LIN {X 0,Y 496.716,Z 59.924,A -85,B 0,C 180,E1 24096.26,E2 24096.26} C_VEL
LIN {X 0,Y 496.76,Z 59.921,A -85,B 0,C 180,E1 24092.813,E2 24092.813} C_VEL
LIN {X 0,Y 496.725,Z 59.923,A -85,B 0,C 180,E1 24089.385,E2 24089.385} C_VEL
LIN {X 0,Y 496.699,Z 59.924,A -85,B 0,C 180,E1 24085.971,E2 24085.971} C_VEL
LIN {X 0,Y 496.701,Z 59.924,A -85,B 0,C 180,E1 24082.415,E2 24082.415} C_VEL
LIN {X 0,Y 496.743,Z 59.924,A -85,B 0,C 180,E1 24079.009,E2 24079.009} C_VEL
LIN {X 0,Y 496.74,Z 59.919,A -85,B 0,C 180,E1 24075.443,E2 24075.443} C_VEL
LIN {X 0,Y 496.703,Z 59.927,A -85,B 0,C 180,E1 24072.03,E2 24072.03} C_VEL
LIN {X 0,Y 496.702,Z 59.928,A -85,B 0,C 180,E1 24068.611,E2 24068.611} C_VEL
LIN {X 0,Y 496.775,Z 60.152,A -85,B 0,C 180,E1 24065.671,E2 24065.671} C_VEL
LIN {X 0,Y 502.744,Z 77.218,A -85,B 0,C 180,E1 24063.56,E2 24063.56} C_VEL
LIN {X 0,Y 505.317,Z 85.52,A -85,B 0,C 180,E1 24062.629,E2 24062.629} C_VEL
LIN {X 0,Y 502.906,Z 130.198,A -85,B 0,C 180,E1 24058.89,E2 24058.89} C_VEL
LIN {X 0,Y 501.717,Z 159.661,A -85,B 0,C 180,E1 24056.536,E2 24056.536} C_VEL
LIN {X 0,Y 503.214,Z 173.732,A -85,B 0,C 180,E1 24056.253,E2 24056.253} C_VEL
LIN {X 0,Y 501.873,Z 362.743,A -85,B 0,C 180,E1 24053.517,E2 24053.517} C_VEL
LIN {X 0,Y 501.376,Z 381.426,A -85,B 0,C 180,E1 24053.042,E2 24053.042} C_VEL
LIN {X 0,Y 500.757,Z 399.797,A -85,B 0,C 180,E1 24052.357,E2 24052.357} C_VEL
LIN {X 0,Y 500.08,Z 416.685,A -85,B 0,C 180,E1 24051.524,E2 24051.524} C_VEL
LIN {X 0,Y 499.326,Z 433.862,A -85,B 0,C 180,E1 24050.452,E2 24050.452} C_VEL
LIN {X 0,Y 498.576,Z 450.092,A -85,B 0,C 180,E1 24049.202,E2 24049.202} C_VEL
LIN {X 0,Y 497.872,Z 465.754,A -85,B 0,C 180,E1 24047.733,E2 24047.733} C_VEL
LIN {X 0,Y 497.273,Z 480.092,A -85,B 0,C 180,E1 24046.11,E2 24046.11} C_VEL
LIN {X 0,Y 496.822,Z 492.31,A -85,B 0,C 180,E1 24044.452,E2 24044.452} C_VEL
LIN {X 0,Y 496.496,Z 503.201,A -85,B 0,C 180,E1 24042.681,E2 24042.681} C_VEL
LIN {X 0,Y 496.273,Z 512.736,A -85,B 0,C 180,E1 24040.8,E2 24040.8} C_VEL
LIN {X 0,Y 496.163,Z 520.846,A -85,B 0,C 180,E1 24038.81,E2 24038.81} C_VEL
LIN {X 0,Y 496.121,Z 527.106,A -85,B 0,C 180,E1 24036.83,E2 24036.83} C_VEL
LIN {X 0,Y 496.12,Z 531.896,A -85,B 0,C 180,E1 24034.741,E2 24034.741} C_VEL
LIN {X 0,Y 496.135,Z 534.912,A -85,B 0,C 180,E1 24032.658,E2 24032.658} C_VEL
LIN {X 0,Y 496.149,Z 536.233,A -85,B 0,C 180,E1 24030.578,E2 24030.578} C_VEL
LIN {X 0,Y 496.141,Z 535.884,A -85,B 0,C 180,E1 24028.5,E2 24028.5} C_VEL
LIN {X 0,Y 496.114,Z 533.857,A -85,B 0,C 180,E1 24026.419,E2 24026.419} C_VEL
LIN {X 0,Y 496.098,Z 530.107,A -85,B 0,C 180,E1 24024.333,E2 24024.333} C_VEL
LIN {X 0,Y 496.123,Z 524.542,A -85,B 0,C 180,E1 24022.241,E2 24022.241} C_VEL
LIN {X 0,Y 496.195,Z 517.201,A -85,B 0,C 180,E1 24020.184,E2 24020.184} C_VEL
LIN {X 0,Y 496.361,Z 508.369,A -85,B 0,C 180,E1 24018.233,E2 24018.233} C_VEL
LIN {X 0,Y 496.659,Z 498.035,A -85,B 0,C 180,E1 24016.378,E2 24016.378} C_VEL
LIN {X 0,Y 497.07,Z 486.087,A -85,B 0,C 180,E1 24014.603,E2 24014.603} C_VEL
LIN {X 0,Y 497.658,Z 472.121,A -85,B 0,C 180,E1 24012.883,E2 24012.883} C_VEL
LIN {X 0,Y 498.316,Z 457.588,A -85,B 0,C 180,E1 24011.397,E2 24011.397} C_VEL
LIN {X 0,Y 499.047,Z 442.169,A -85,B 0,C 180,E1 24010.088,E2 24010.088} C_VEL
LIN {X 0,Y 499.804,Z 425.94,A -85,B 0,C 180,E1 24008.957,E2 24008.957} C_VEL
LIN {X 0,Y 500.54,Z 408.959,A -85,B 0,C 180,E1 24008.005,E2 24008.005} C_VEL
LIN {X 0,Y 501.216,Z 391.162,A -85,B 0,C 180,E1 24007.233,E2 24007.233} C_VEL
LIN {X 0,Y 501.791,Z 372.509,A -85,B 0,C 180,E1 24006.648,E2 24006.648} C_VEL
LIN {X 0,Y 502.171,Z 353.099,A -85,B 0,C 180,E1 24006.264,E2 24006.264} C_VEL
LIN {X 0,Y 503.355,Z 163.342,A -85,B 0,C 180,E1 24003.523,E2 24003.523} C_VEL
LIN {X 0,Y 502.895,Z 155.431,A -85,B 0,C 180,E1 24003.364,E2 24003.364} C_VEL
LIN {X 0,Y 505.189,Z 81.94,A -85,B 0,C 180,E1 23999.846,E2 23999.846} C_VEL
LIN {X 0,Y 496.866,Z 60.542,A -85,B 0,C 180,E1 23998.232,E2 23998.232} C_VEL
LIN {X 0,Y 496.764,Z 59.943,A -85,B 0,C 180,E1 23998.04,E2 23998.04} C_VEL
LIN {X 0,Y 496.765,Z 59.917,A -85,B 0,C 180,E1 23994.404,E2 23994.404} C_VEL
LIN {X 0,Y 496.767,Z 59.917,A -85,B 0,C 180,E1 23990.796,E2 23990.796} C_VEL
LIN {X 0,Y 496.755,Z 59.92,A -85,B 0,C 180,E1 23987.279,E2 23987.279} C_VEL
LIN {X 0,Y 496.762,Z 59.919,A -85,B 0,C 180,E1 23983.735,E2 23983.735} C_VEL
LIN {X 0,Y 496.767,Z 59.918,A -85,B 0,C 180,E1 23980.247,E2 23980.247} C_VEL
LIN {X 0,Y 496.768,Z 59.916,A -85,B 0,C 180,E1 23976.711,E2 23976.711} C_VEL
LIN {X 0,Y 496.761,Z 59.915,A -85,B 0,C 180,E1 23973.146,E2 23973.146} C_VEL
LIN {X 0,Y 496.749,Z 59.917,A -85,B 0,C 180,E1 23969.599,E2 23969.599} C_VEL
LIN {X 0,Y 496.754,Z 59.92,A -85,B 0,C 180,E1 23966.026,E2 23966.026} C_VEL
LIN {X 0,Y 496.774,Z 59.916,A -85,B 0,C 180,E1 23962.483,E2 23962.483} C_VEL
LIN {X 0,Y 496.77,Z 59.913,A -85,B 0,C 180,E1 23958.908,E2 23958.908} C_VEL
LIN {X 0,Y 496.768,Z 59.913,A -85,B 0,C 180,E1 23955.288,E2 23955.288} C_VEL
LIN {X 0,Y 496.746,Z 59.917,A -85,B 0,C 180,E1 23951.729,E2 23951.729} C_VEL
LIN {X 0,Y 496.742,Z 59.918,A -85,B 0,C 180,E1 23948.216,E2 23948.216} C_VEL
LIN {X 0,Y 496.761,Z 59.915,A -85,B 0,C 180,E1 23944.733,E2 23944.733} C_VEL
LIN {X 0,Y 496.773,Z 59.918,A -85,B 0,C 180,E1 23941.153,E2 23941.153} C_VEL
LIN {X 0,Y 496.763,Z 59.916,A -85,B 0,C 180,E1 23937.577,E2 23937.577} C_VEL
LIN {X 0,Y 496.737,Z 59.916,A -85,B 0,C 180,E1 23934.108,E2 23934.108} C_VEL
LIN {X 0,Y 496.732,Z 59.915,A -85,B 0,C 180,E1 23930.499,E2 23930.499} C_VEL
LIN {X 0,Y 496.748,Z 59.917,A -85,B 0,C 180,E1 23926.971,E2 23926.971} C_VEL
LIN {X 0,Y 496.772,Z 59.919,A -85,B 0,C 180,E1 23923.513,E2 23923.513} C_VEL
LIN {X 0,Y 496.754,Z 59.917,A -85,B 0,C 180,E1 23919.99,E2 23919.99} C_VEL
LIN {X 0,Y 496.729,Z 59.902,A -85,B 0,C 180,E1 23916.512,E2 23916.512} C_VEL
LIN {X 0,Y 496.728,Z 59.921,A -85,B 0,C 180,E1 23912.94,E2 23912.94} C_VEL
LIN {X 0,Y 496.754,Z 59.91,A -85,B 0,C 180,E1 23909.479,E2 23909.479} C_VEL
LIN {X 0,Y 496.768,Z 59.92,A -85,B 0,C 180,E1 23905.976,E2 23905.976} C_VEL
LIN {X 0,Y 496.741,Z 59.92,A -85,B 0,C 180,E1 23902.418,E2 23902.418} C_VEL
LIN {X 0,Y 496.719,Z 59.919,A -85,B 0,C 180,E1 23898.988,E2 23898.988} C_VEL
LIN {X 0,Y 496.724,Z 59.923,A -85,B 0,C 180,E1 23895.442,E2 23895.442} C_VEL
LIN {X 0,Y 496.765,Z 59.919,A -85,B 0,C 180,E1 23892.037,E2 23892.037} C_VEL
LIN {X 0,Y 496.741,Z 59.922,A -85,B 0,C 180,E1 23888.605,E2 23888.605} C_VEL
LIN {X 0,Y 496.76,Z 59.922,A -85,B 0,C 180,E1 23886.138,E2 23886.138} C_VEL
LIN {X 0,Y 496.526,Z 60.974,A -85,B 0,C 180,E1 23885.641,E2 23885.641} C_VEL
LIN {X 0,Y 495.866,Z 64.234,A -85,B 0,C 180,E1 23885.105,E2 23885.105} C_VEL
LIN {X 0,Y 493.642,Z 74.787,A -85,B 0,C 180,E1 23884.064,E2 23884.064} C_VEL
LIN {X 0,Y 492.439,Z 83.383,A -85,B 0,C 180,E1 23883.217,E2 23883.217} C_VEL
LIN {X 0,Y 492.424,Z 84.219,A -85,B 0,C 180,E1 23883.128,E2 23883.128} C_VEL
LIN {X 0,Y 492.207,Z 114.606,A -85,B 0,C 180,E1 23879.841,E2 23879.841} C_VEL
LIN {X 0,Y 491.855,Z 147.091,A -85,B 0,C 180,E1 23876.3,E2 23876.3} C_VEL
LIN {X 0,Y 491.542,Z 180.424,A -85,B 0,C 180,E1 23872.735,E2 23872.735} C_VEL
LIN {X 0,Y 491.569,Z 185.791,A -85,B 0,C 180,E1 23872.215,E2 23872.215} C_VEL
LIN {X 0,Y 492.039,Z 191.108,A -85,B 0,C 180,E1 23872.114,E2 23872.114} C_VEL
LIN {X 0,Y 491.357,Z 297.481,A -85,B 0,C 180,E1 23870.513,E2 23870.513} C_VEL
LIN {X 0,Y 491.296,Z 311.859,A -85,B 0,C 180,E1 23870.086,E2 23870.086} C_VEL
LIN {X 0,Y 491.08,Z 325.962,A -85,B 0,C 180,E1 23869.449,E2 23869.449} C_VEL
LIN {X 0,Y 490.712,Z 339.55,A -85,B 0,C 180,E1 23868.594,E2 23868.594} C_VEL
LIN {X 0,Y 490.308,Z 351.863,A -85,B 0,C 180,E1 23867.565,E2 23867.565} C_VEL
LIN {X 0,Y 489.912,Z 362.623,A -85,B 0,C 180,E1 23866.417,E2 23866.417} C_VEL
LIN {X 0,Y 489.49,Z 372.793,A -85,B 0,C 180,E1 23865.034,E2 23865.034} C_VEL
LIN {X 0,Y 489.123,Z 381.598,A -85,B 0,C 180,E1 23863.475,E2 23863.475} C_VEL
LIN {X 0,Y 488.845,Z 388.636,A -85,B 0,C 180,E1 23861.801,E2 23861.801} C_VEL
LIN {X 0,Y 488.666,Z 393.601,A -85,B 0,C 180,E1 23860.134,E2 23860.134} C_VEL
LIN {X 0,Y 488.558,Z 396.808,A -85,B 0,C 180,E1 23858.472,E2 23858.472} C_VEL
LIN {X 0,Y 488.503,Z 398.475,A -85,B 0,C 180,E1 23856.581,E2 23856.581} C_VEL
LIN {X 0,Y 488.508,Z 398.105,A -85,B 0,C 180,E1 23854.695,E2 23854.695} C_VEL
LIN {X 0,Y 488.575,Z 395.704,A -85,B 0,C 180,E1 23852.814,E2 23852.814} C_VEL
LIN {X 0,Y 488.708,Z 391.51,A -85,B 0,C 180,E1 23851.054,E2 23851.054} C_VEL
LIN {X 0,Y 488.893,Z 386.21,A -85,B 0,C 180,E1 23849.53,E2 23849.53} C_VEL
LIN {X 0,Y 489.189,Z 378.47,A -85,B 0,C 180,E1 23847.891,E2 23847.891} C_VEL
LIN {X 0,Y 489.571,Z 368.931,A -85,B 0,C 180,E1 23846.369,E2 23846.369} C_VEL
LIN {X 0,Y 489.993,Z 357.955,A -85,B 0,C 180,E1 23845.024,E2 23845.024} C_VEL
LIN {X 0,Y 490.361,Z 346.306,A -85,B 0,C 180,E1 23843.913,E2 23843.913} C_VEL
LIN {X 0,Y 490.725,Z 334.558,A -85,B 0,C 180,E1 23843.036,E2 23843.036} C_VEL
LIN {X 0,Y 491.017,Z 321.028,A -85,B 0,C 180,E1 23842.276,E2 23842.276} C_VEL
LIN {X 0,Y 491.145,Z 306.68,A -85,B 0,C 180,E1 23841.707,E2 23841.707} C_VEL
LIN {X 0,Y 491.164,Z 291.861,A -85,B 0,C 180,E1 23841.346,E2 23841.346} C_VEL
LIN {X 0,Y 491.891,Z 181.867,A -85,B 0,C 180,E1 23839.725,E2 23839.725} C_VEL
LIN {X 0,Y 492.368,Z 131.209,A -85,B 0,C 180,E1 23836.494,E2 23836.494} C_VEL
LIN {X 0,Y 492.96,Z 86.133,A -85,B 0,C 180,E1 23833.533,E2 23833.533} C_VEL
LIN {X 0,Y 493.461,Z 85.428,A -85,B 0,C 180,E1 23833.338,E2 23833.338} C_VEL
LIN {X 0,Y 495.053,Z 86.354,A -85,B 0,C 180,E1 23833.122,E2 23833.122} C_VEL
LIN {X 0,Y 493.208,Z 136.927,A -85,B 0,C 180,E1 23829.406,E2 23829.406} C_VEL
LIN {X 0,Y 492.18,Z 171.769,A -85,B 0,C 180,E1 23826.9,E2 23826.9} C_VEL
LIN {X 0,Y 493.337,Z 184.723,A -85,B 0,C 180,E1 23826.64,E2 23826.64} C_VEL
LIN {X 0,Y 492.138,Z 292.661,A -85,B 0,C 180,E1 23824.909,E2 23824.909} C_VEL
LIN {X 0,Y 491.908,Z 307.221,A -85,B 0,C 180,E1 23824.474,E2 23824.474} C_VEL
LIN {X 0,Y 491.557,Z 320.784,A -85,B 0,C 180,E1 23823.872,E2 23823.872} C_VEL
LIN {X 0,Y 491.096,Z 334.583,A -85,B 0,C 180,E1 23823.043,E2 23823.043} C_VEL
LIN {X 0,Y 490.581,Z 347.204,A -85,B 0,C 180,E1 23822.045,E2 23822.045} C_VEL
LIN {X 0,Y 490.103,Z 358.821,A -85,B 0,C 180,E1 23820.879,E2 23820.879} C_VEL
LIN {X 0,Y 489.623,Z 369.502,A -85,B 0,C 180,E1 23819.516,E2 23819.516} C_VEL
LIN {X 0,Y 489.213,Z 378.649,A -85,B 0,C 180,E1 23818.015,E2 23818.015} C_VEL
LIN {X 0,Y 488.922,Z 385.866,A -85,B 0,C 180,E1 23816.484,E2 23816.484} C_VEL
LIN {X 0,Y 488.704,Z 391.966,A -85,B 0,C 180,E1 23814.72,E2 23814.72} C_VEL
LIN {X 0,Y 488.576,Z 396.002,A -85,B 0,C 180,E1 23812.952,E2 23812.952} C_VEL
LIN {X 0,Y 488.519,Z 398.188,A -85,B 0,C 180,E1 23811.222,E2 23811.222} C_VEL
LIN {X 0,Y 488.523,Z 398.654,A -85,B 0,C 180,E1 23809.394,E2 23809.394} C_VEL
LIN {X 0,Y 488.582,Z 397.307,A -85,B 0,C 180,E1 23807.627,E2 23807.627} C_VEL
LIN {X 0,Y 488.713,Z 394.286,A -85,B 0,C 180,E1 23805.899,E2 23805.899} C_VEL
LIN {X 0,Y 488.92,Z 389.202,A -85,B 0,C 180,E1 23804.126,E2 23804.126} C_VEL
LIN {X 0,Y 489.201,Z 382.95,A -85,B 0,C 180,E1 23802.573,E2 23802.573} C_VEL
LIN {X 0,Y 489.611,Z 374.598,A -85,B 0,C 180,E1 23801.001,E2 23801.001} C_VEL
LIN {X 0,Y 490.115,Z 364.396,A -85,B 0,C 180,E1 23799.531,E2 23799.531} C_VEL
LIN {X 0,Y 490.644,Z 353.329,A -85,B 0,C 180,E1 23798.281,E2 23798.281} C_VEL
LIN {X 0,Y 491.202,Z 341.189,A -85,B 0,C 180,E1 23797.197,E2 23797.197} C_VEL
LIN {X 0,Y 491.738,Z 327.186,A -85,B 0,C 180,E1 23796.241,E2 23796.241} C_VEL
LIN {X 0,Y 492.164,Z 313.062,A -85,B 0,C 180,E1 23795.523,E2 23795.523} C_VEL
LIN {X 0,Y 492.489,Z 297.592,A -85,B 0,C 180,E1 23794.979,E2 23794.979} C_VEL
LIN {X 0,Y 492.743,Z 277.093,A -85,B 0,C 180,E1 23794.576,E2 23794.576} C_VEL
LIN {X 0,Y 493.812,Z 188.367,A -85,B 0,C 180,E1 23793.093,E2 23793.093} C_VEL
LIN {X 0,Y 491.269,Z 174.322,A -85,B 0,C 180,E1 23792.689,E2 23792.689} C_VEL
LIN {X 0,Y 492.482,Z 144.862,A -85,B 0,C 180,E1 23789.028,E2 23789.028} C_VEL
LIN {X 0,Y 493.866,Z 117.28,A -85,B 0,C 180,E1 23785.546,E2 23785.546} C_VEL
LIN {X 0,Y 495.5,Z 87.632,A -85,B 0,C 180,E1 23781.733,E2 23781.733} C_VEL
LIN {X 0,Y 495.539,Z 84.368,A -85,B 0,C 180,E1 23781.297,E2 23781.297} C_VEL
LIN {X 0,Y 491.064,Z 68.425,A -85,B 0,C 180,E1 23778.766,E2 23778.766} C_VEL
LIN {X 0,Y 488.818,Z 61.026,A -85,B 0,C 180,E1 23777.483,E2 23777.483} C_VEL
LIN {X 0,Y 488.832,Z 60.909,A -85,B 0,C 180,E1 23773.967,E2 23773.967} C_VEL
LIN {X 0,Y 488.822,Z 60.908,A -85,B 0,C 180,E1 23770.37,E2 23770.37} C_VEL
LIN {X 0,Y 488.787,Z 60.91,A -85,B 0,C 180,E1 23766.932,E2 23766.932} C_VEL
LIN {X 0,Y 488.781,Z 60.912,A -85,B 0,C 180,E1 23763.381,E2 23763.381} C_VEL
LIN {X 0,Y 488.797,Z 60.911,A -85,B 0,C 180,E1 23759.883,E2 23759.883} C_VEL
LIN {X 0,Y 488.824,Z 60.91,A -85,B 0,C 180,E1 23756.365,E2 23756.365} C_VEL
LIN {X 0,Y 488.807,Z 60.91,A -85,B 0,C 180,E1 23752.832,E2 23752.832} C_VEL
LIN {X 0,Y 488.774,Z 60.911,A -85,B 0,C 180,E1 23749.391,E2 23749.391} C_VEL
LIN {X 0,Y 488.77,Z 60.91,A -85,B 0,C 180,E1 23745.79,E2 23745.79} C_VEL
LIN {X 0,Y 488.799,Z 60.91,A -85,B 0,C 180,E1 23742.378,E2 23742.378} C_VEL
LIN {X 0,Y 488.827,Z 60.908,A -85,B 0,C 180,E1 23738.775,E2 23738.775} C_VEL
LIN {X 0,Y 488.79,Z 60.911,A -85,B 0,C 180,E1 23735.263,E2 23735.263} C_VEL
LIN {X 0,Y 488.765,Z 60.912,A -85,B 0,C 180,E1 23731.8,E2 23731.8} C_VEL
LIN {X 0,Y 488.761,Z 60.913,A -85,B 0,C 180,E1 23728.144,E2 23728.144} C_VEL
LIN {X 0,Y 488.787,Z 60.913,A -85,B 0,C 180,E1 23724.705,E2 23724.705} C_VEL
LIN {X 0,Y 488.816,Z 60.912,A -85,B 0,C 180,E1 23721.199,E2 23721.199} C_VEL
LIN {X 0,Y 488.765,Z 60.915,A -85,B 0,C 180,E1 23717.777,E2 23717.777} C_VEL
LIN {X 0,Y 488.758,Z 60.915,A -85,B 0,C 180,E1 23714.275,E2 23714.275} C_VEL
LIN {X 0,Y 488.77,Z 60.915,A -85,B 0,C 180,E1 23710.736,E2 23710.736} C_VEL
LIN {X 0,Y 488.817,Z 60.908,A -85,B 0,C 180,E1 23707.41,E2 23707.41} C_VEL
LIN {X 0,Y 488.795,Z 61.141,A -85,B 0,C 180,E1 23706.24,E2 23706.24} C_VEL
LIN {X 0,Y 494.085,Z 75.723,A -85,B 0,C 180,E1 23704.345,E2 23704.345} C_VEL
LIN {X 0,Y 498.039,Z 88.036,A -85,B 0,C 180,E1 23702.899,E2 23702.899} C_VEL
LIN {X 0,Y 495.366,Z 133.317,A -85,B 0,C 180,E1 23699.041,E2 23699.041} C_VEL
LIN {X 0,Y 494.195,Z 159.804,A -85,B 0,C 180,E1 23696.886,E2 23696.886} C_VEL
LIN {X 0,Y 495.772,Z 174.654,A -85,B 0,C 180,E1 23696.58,E2 23696.58} C_VEL
LIN {X 0,Y 494.31,Z 362.064,A -85,B 0,C 180,E1 23693.828,E2 23693.828} C_VEL
LIN {X 0,Y 493.779,Z 380.78,A -85,B 0,C 180,E1 23693.345,E2 23693.345} C_VEL
LIN {X 0,Y 493.115,Z 398.948,A -85,B 0,C 180,E1 23692.66,E2 23692.66} C_VEL
LIN {X 0,Y 492.342,Z 416.524,A -85,B 0,C 180,E1 23691.776,E2 23691.776} C_VEL
LIN {X 0,Y 491.555,Z 433.003,A -85,B 0,C 180,E1 23690.728,E2 23690.728} C_VEL
LIN {X 0,Y 490.75,Z 449.218,A -85,B 0,C 180,E1 23689.459,E2 23689.459} C_VEL
LIN {X 0,Y 489.979,Z 465.054,A -85,B 0,C 180,E1 23687.947,E2 23687.947} C_VEL
LIN {X 0,Y 489.363,Z 478.705,A -85,B 0,C 180,E1 23686.378,E2 23686.378} C_VEL
LIN {X 0,Y 488.868,Z 491.134,A -85,B 0,C 180,E1 23684.669,E2 23684.669} C_VEL
LIN {X 0,Y 488.526,Z 501.928,A -85,B 0,C 180,E1 23682.891,E2 23682.891} C_VEL
LIN {X 0,Y 488.294,Z 511.506,A -85,B 0,C 180,E1 23680.979,E2 23680.979} C_VEL
LIN {X 0,Y 488.195,Z 519.655,A -85,B 0,C 180,E1 23678.955,E2 23678.955} C_VEL
LIN {X 0,Y 488.165,Z 525.946,A -85,B 0,C 180,E1 23676.942,E2 23676.942} C_VEL
LIN {X 0,Y 488.18,Z 530.761,A -85,B 0,C 180,E1 23674.818,E2 23674.818} C_VEL
LIN {X 0,Y 488.206,Z 533.796,A -85,B 0,C 180,E1 23672.701,E2 23672.701} C_VEL
LIN {X 0,Y 488.225,Z 535.128,A -85,B 0,C 180,E1 23670.588,E2 23670.588} C_VEL
LIN {X 0,Y 488.215,Z 534.781,A -85,B 0,C 180,E1 23668.475,E2 23668.475} C_VEL
LIN {X 0,Y 488.179,Z 532.751,A -85,B 0,C 180,E1 23666.361,E2 23666.361} C_VEL
LIN {X 0,Y 488.15,Z 528.992,A -85,B 0,C 180,E1 23664.241,E2 23664.241} C_VEL
LIN {X 0,Y 488.156,Z 523.411,A -85,B 0,C 180,E1 23662.113,E2 23662.113} C_VEL
LIN {X 0,Y 488.214,Z 516.331,A -85,B 0,C 180,E1 23660.091,E2 23660.091} C_VEL
LIN {X 0,Y 488.385,Z 507.338,A -85,B 0,C 180,E1 23658.068,E2 23658.068} C_VEL
LIN {X 0,Y 488.697,Z 496.822,A -85,B 0,C 180,E1 23656.151,E2 23656.151} C_VEL
LIN {X 0,Y 489.158,Z 484.562,A -85,B 0,C 180,E1 23654.311,E2 23654.311} C_VEL
LIN {X 0,Y 489.791,Z 470.803,A -85,B 0,C 180,E1 23652.6,E2 23652.6} C_VEL
LIN {X 0,Y 490.509,Z 456.185,A -85,B 0,C 180,E1 23651.09,E2 23651.09} C_VEL
LIN {X 0,Y 491.31,Z 440.484,A -85,B 0,C 180,E1 23649.747,E2 23649.747} C_VEL
LIN {X 0,Y 492.172,Z 423.339,A -85,B 0,C 180,E1 23648.552,E2 23648.552} C_VEL
LIN {X 0,Y 492.983,Z 405.873,A -85,B 0,C 180,E1 23647.587,E2 23647.587} C_VEL
LIN {X 0,Y 493.729,Z 387.328,A -85,B 0,C 180,E1 23646.811,E2 23646.811} C_VEL
LIN {X 0,Y 494.323,Z 368.66,A -85,B 0,C 180,E1 23646.26,E2 23646.26} C_VEL
LIN {X 0,Y 494.652,Z 348.014,A -85,B 0,C 180,E1 23645.887,E2 23645.887} C_VEL
LIN {X 0,Y 495.912,Z 163.899,A -85,B 0,C 180,E1 23643.19,E2 23643.19} C_VEL
LIN {X 0,Y 495.447,Z 155.03,A -85,B 0,C 180,E1 23642.996,E2 23642.996} C_VEL
LIN {X 0,Y 497.86,Z 84.428,A -85,B 0,C 180,E1 23639.555,E2 23639.555} C_VEL
LIN {X 0,Y 488.912,Z 61.44,A -85,B 0,C 180,E1 23637.776,E2 23637.776} C_VEL
LIN {X 0,Y 488.832,Z 60.926,A -85,B 0,C 180,E1 23637.597,E2 23637.597} C_VEL
LIN {X 0,Y 488.823,Z 60.909,A -85,B 0,C 180,E1 23634.054,E2 23634.054} C_VEL
LIN {X 0,Y 488.83,Z 60.907,A -85,B 0,C 180,E1 23630.454,E2 23630.454} C_VEL
LIN {X 0,Y 488.823,Z 60.906,A -85,B 0,C 180,E1 23626.905,E2 23626.905} C_VEL
LIN {X 0,Y 488.815,Z 60.907,A -85,B 0,C 180,E1 23623.268,E2 23623.268} C_VEL
LIN {X 0,Y 488.816,Z 60.909,A -85,B 0,C 180,E1 23619.657,E2 23619.657} C_VEL
LIN {X 0,Y 488.828,Z 60.908,A -85,B 0,C 180,E1 23616.092,E2 23616.092} C_VEL
LIN {X 0,Y 488.828,Z 60.907,A -85,B 0,C 180,E1 23612.544,E2 23612.544} C_VEL
LIN {X 0,Y 488.833,Z 60.903,A -85,B 0,C 180,E1 23608.908,E2 23608.908} C_VEL
LIN {X 0,Y 488.82,Z 60.904,A -85,B 0,C 180,E1 23605.303,E2 23605.303} C_VEL
LIN {X 0,Y 488.807,Z 60.907,A -85,B 0,C 180,E1 23601.73,E2 23601.73} C_VEL
LIN {X 0,Y 488.809,Z 60.908,A -85,B 0,C 180,E1 23598.114,E2 23598.114} C_VEL
LIN {X 0,Y 488.831,Z 60.903,A -85,B 0,C 180,E1 23594.571,E2 23594.571} C_VEL
LIN {X 0,Y 488.831,Z 60.907,A -85,B 0,C 180,E1 23590.959,E2 23590.959} C_VEL
LIN {X 0,Y 488.835,Z 60.903,A -85,B 0,C 180,E1 23587.285,E2 23587.285} C_VEL
LIN {X 0,Y 488.809,Z 60.902,A -85,B 0,C 180,E1 23583.753,E2 23583.753} C_VEL
LIN {X 0,Y 488.798,Z 60.901,A -85,B 0,C 180,E1 23580.234,E2 23580.234} C_VEL
LIN {X 0,Y 488.81,Z 60.908,A -85,B 0,C 180,E1 23576.716,E2 23576.716} C_VEL
LIN {X 0,Y 488.838,Z 60.907,A -85,B 0,C 180,E1 23573.187,E2 23573.187} C_VEL
LIN {X 0,Y 488.828,Z 60.9,A -85,B 0,C 180,E1 23569.63,E2 23569.63} C_VEL
LIN {X 0,Y 488.798,Z 60.902,A -85,B 0,C 180,E1 23566.153,E2 23566.153} C_VEL
LIN {X 0,Y 488.791,Z 60.905,A -85,B 0,C 180,E1 23562.623,E2 23562.623} C_VEL
LIN {X 0,Y 488.807,Z 60.907,A -85,B 0,C 180,E1 23559.15,E2 23559.15} C_VEL
LIN {X 0,Y 488.831,Z 60.889,A -85,B 0,C 180,E1 23555.724,E2 23555.724} C_VEL
LIN {X 0,Y 488.808,Z 60.907,A -85,B 0,C 180,E1 23552.2,E2 23552.2} C_VEL
LIN {X 0,Y 488.784,Z 60.904,A -85,B 0,C 180,E1 23548.763,E2 23548.763} C_VEL
LIN {X 0,Y 488.788,Z 60.903,A -85,B 0,C 180,E1 23545.199,E2 23545.199} C_VEL
LIN {X 0,Y 488.818,Z 60.912,A -85,B 0,C 180,E1 23541.7,E2 23541.7} C_VEL
LIN {X 0,Y 488.83,Z 60.907,A -85,B 0,C 180,E1 23538.116,E2 23538.116} C_VEL
LIN {X 0,Y 488.802,Z 60.91,A -85,B 0,C 180,E1 23534.555,E2 23534.555} C_VEL
LIN {X 0,Y 488.775,Z 60.913,A -85,B 0,C 180,E1 23531.043,E2 23531.043} C_VEL
LIN {X 0,Y 488.777,Z 60.916,A -85,B 0,C 180,E1 23527.411,E2 23527.411} C_VEL
LIN {X 0,Y 488.827,Z 61.168,A -85,B 0,C 180,E1 23525.781,E2 23525.781} C_VEL
LIN {X 0,Y 492.431,Z 75.428,A -85,B 0,C 180,E1 23524.062,E2 23524.062} C_VEL
LIN {X 0,Y 492.424,Z 84.219,A -85,B 0,C 180,E1 23523.128,E2 23523.128} C_VEL
LIN {X 0,Y 491.471,Z 90.111,A -85,B 0,C 180,E1 23522.55,E2 23522.55} C_VEL
LIN {X 0,Y 485.216,Z 107.25,A -85,B 0,C 180,E1 23521.027,E2 23521.027} C_VEL
LIN {X 0,Y 484.662,Z 111.429,A -85,B 0,C 180,E1 23520.597,E2 23520.597} C_VEL
LIN {X 0,Y 484.302,Z 143.545,A -85,B 0,C 180,E1 23517.078,E2 23517.078} C_VEL
LIN {X 0,Y 483.926,Z 176.363,A -85,B 0,C 180,E1 23513.548,E2 23513.548} C_VEL
LIN {X 0,Y 483.915,Z 186.439,A -85,B 0,C 180,E1 23512.511,E2 23512.511} C_VEL
LIN {X 0,Y 484.433,Z 191.716,A -85,B 0,C 180,E1 23512.399,E2 23512.399} C_VEL
LIN {X 0,Y 483.702,Z 298.42,A -85,B 0,C 180,E1 23510.77,E2 23510.77} C_VEL
LIN {X 0,Y 483.639,Z 312.821,A -85,B 0,C 180,E1 23510.338,E2 23510.338} C_VEL
LIN {X 0,Y 483.415,Z 326.772,A -85,B 0,C 180,E1 23509.701,E2 23509.701} C_VEL
LIN {X 0,Y 483.024,Z 340.331,A -85,B 0,C 180,E1 23508.838,E2 23508.838} C_VEL
LIN {X 0,Y 482.586,Z 352.724,A -85,B 0,C 180,E1 23507.793,E2 23507.793} C_VEL
LIN {X 0,Y 482.156,Z 363.533,A -85,B 0,C 180,E1 23506.628,E2 23506.628} C_VEL
LIN {X 0,Y 481.712,Z 373.35,A -85,B 0,C 180,E1 23505.283,E2 23505.283} C_VEL
LIN {X 0,Y 481.322,Z 381.658,A -85,B 0,C 180,E1 23503.82,E2 23503.82} C_VEL
LIN {X 0,Y 481.02,Z 388.542,A -85,B 0,C 180,E1 23502.24,E2 23502.24} C_VEL
LIN {X 0,Y 480.803,Z 393.911,A -85,B 0,C 180,E1 23500.544,E2 23500.544} C_VEL
LIN {X 0,Y 480.656,Z 397.602,A -85,B 0,C 180,E1 23498.733,E2 23498.733} C_VEL
LIN {X 0,Y 480.585,Z 399.41,A -85,B 0,C 180,E1 23496.93,E2 23496.93} C_VEL
LIN {X 0,Y 480.573,Z 399.446,A -85,B 0,C 180,E1 23495.132,E2 23495.132} C_VEL
LIN {X 0,Y 480.626,Z 397.72,A -85,B 0,C 180,E1 23493.338,E2 23493.338} C_VEL
LIN {X 0,Y 480.762,Z 393.835,A -85,B 0,C 180,E1 23491.429,E2 23491.429} C_VEL
LIN {X 0,Y 480.972,Z 388.092,A -85,B 0,C 180,E1 23489.642,E2 23489.642} C_VEL
LIN {X 0,Y 481.251,Z 381.205,A -85,B 0,C 180,E1 23488.094,E2 23488.094} C_VEL
LIN {X 0,Y 481.607,Z 372.979,A -85,B 0,C 180,E1 23486.667,E2 23486.667} C_VEL
LIN {X 0,Y 482.053,Z 362.367,A -85,B 0,C 180,E1 23485.24,E2 23485.24} C_VEL
LIN {X 0,Y 482.488,Z 350.344,A -85,B 0,C 180,E1 23483.992,E2 23483.992} C_VEL
LIN {X 0,Y 482.896,Z 337.65,A -85,B 0,C 180,E1 23482.982,E2 23482.982} C_VEL
LIN {X 0,Y 483.224,Z 324.858,A -85,B 0,C 180,E1 23482.21,E2 23482.21} C_VEL
LIN {X 0,Y 483.395,Z 310.077,A -85,B 0,C 180,E1 23481.569,E2 23481.569} C_VEL
LIN {X 0,Y 483.428,Z 294.303,A -85,B 0,C 180,E1 23481.15,E2 23481.15} C_VEL
LIN {X 0,Y 484.223,Z 182.643,A -85,B 0,C 180,E1 23479.47,E2 23479.47} C_VEL
LIN {X 0,Y 484.725,Z 131.741,A -85,B 0,C 180,E1 23476.216,E2 23476.216} C_VEL
LIN {X 0,Y 485.244,Z 91.93,A -85,B 0,C 180,E1 23473.602,E2 23473.602} C_VEL
LIN {X 0,Y 485.644,Z 90.792,A -85,B 0,C 180,E1 23473.401,E2 23473.401} C_VEL
LIN {X 0,Y 487.281,Z 91.633,A -85,B 0,C 180,E1 23473.151,E2 23473.151} C_VEL
LIN {X 0,Y 486.097,Z 126.624,A -85,B 0,C 180,E1 23470.535,E2 23470.535} C_VEL
LIN {X 0,Y 484.595,Z 171.64,A -85,B 0,C 180,E1 23467.244,E2 23467.244} C_VEL
LIN {X 0,Y 485.839,Z 185.392,A -85,B 0,C 180,E1 23466.959,E2 23466.959} C_VEL
LIN {X 0,Y 484.534,Z 293.233,A -85,B 0,C 180,E1 23465.194,E2 23465.194} C_VEL
LIN {X 0,Y 484.279,Z 308.348,A -85,B 0,C 180,E1 23464.732,E2 23464.732} C_VEL
LIN {X 0,Y 483.841,Z 323.649,A -85,B 0,C 180,E1 23464.019,E2 23464.019} C_VEL
LIN {X 0,Y 483.353,Z 336.654,A -85,B 0,C 180,E1 23463.195,E2 23463.195} C_VEL
LIN {X 0,Y 482.781,Z 350.036,A -85,B 0,C 180,E1 23462.091,E2 23462.091} C_VEL
LIN {X 0,Y 482.221,Z 362.106,A -85,B 0,C 180,E1 23460.801,E2 23460.801} C_VEL
LIN {X 0,Y 481.726,Z 372.155,A -85,B 0,C 180,E1 23459.435,E2 23459.435} C_VEL
LIN {X 0,Y 481.303,Z 381.173,A -85,B 0,C 180,E1 23457.871,E2 23457.871} C_VEL
LIN {X 0,Y 480.971,Z 388.681,A -85,B 0,C 180,E1 23456.142,E2 23456.142} C_VEL
LIN {X 0,Y 480.76,Z 394.129,A -85,B 0,C 180,E1 23454.385,E2 23454.385} C_VEL
LIN {X 0,Y 480.642,Z 397.719,A -85,B 0,C 180,E1 23452.624,E2 23452.624} C_VEL
LIN {X 0,Y 480.596,Z 399.63,A -85,B 0,C 180,E1 23450.709,E2 23450.709} C_VEL
LIN {X 0,Y 480.613,Z 399.554,A -85,B 0,C 180,E1 23448.86,E2 23448.86} C_VEL
LIN {X 0,Y 480.707,Z 397.738,A -85,B 0,C 180,E1 23447.068,E2 23447.068} C_VEL
LIN {X 0,Y 480.886,Z 393.856,A -85,B 0,C 180,E1 23445.182,E2 23445.182} C_VEL
LIN {X 0,Y 481.144,Z 388.336,A -85,B 0,C 180,E1 23443.46,E2 23443.46} C_VEL
LIN {X 0,Y 481.504,Z 381.447,A -85,B 0,C 180,E1 23441.881,E2 23441.881} C_VEL
LIN {X 0,Y 481.984,Z 372.597,A -85,B 0,C 180,E1 23440.334,E2 23440.334} C_VEL
LIN {X 0,Y 482.509,Z 362.89,A -85,B 0,C 180,E1 23439.006,E2 23439.006} C_VEL
LIN {X 0,Y 483.122,Z 351.015,A -85,B 0,C 180,E1 23437.72,E2 23437.72} C_VEL
LIN {X 0,Y 483.735,Z 337.986,A -85,B 0,C 180,E1 23436.627,E2 23436.627} C_VEL
LIN {X 0,Y 484.266,Z 324.406,A -85,B 0,C 180,E1 23435.754,E2 23435.754} C_VEL
LIN {X 0,Y 484.721,Z 309.644,A -85,B 0,C 180,E1 23435.054,E2 23435.054} C_VEL
LIN {X 0,Y 485.039,Z 293.272,A -85,B 0,C 180,E1 23434.545,E2 23434.545} C_VEL
LIN {X 0,Y 486.437,Z 189.597,A -85,B 0,C 180,E1 23432.75,E2 23432.75} C_VEL
LIN {X 0,Y 483.646,Z 174.3,A -85,B 0,C 180,E1 23432.304,E2 23432.304} C_VEL
LIN {X 0,Y 484.989,Z 144.211,A -85,B 0,C 180,E1 23428.514,E2 23428.514} C_VEL
LIN {X 0,Y 486.543,Z 116.166,A -85,B 0,C 180,E1 23424.916,E2 23424.916} C_VEL
LIN {X 0,Y 488.247,Z 87.595,A -85,B 0,C 180,E1 23421.189,E2 23421.189} C_VEL
LIN {X 0,Y 483.953,Z 72.029,A -85,B 0,C 180,E1 23418.677,E2 23418.677} C_VEL
LIN {X 0,Y 480.864,Z 62.019,A -85,B 0,C 180,E1 23416.924,E2 23416.924} C_VEL
LIN {X 0,Y 480.85,Z 61.898,A -85,B 0,C 180,E1 23413.31,E2 23413.31} C_VEL
LIN {X 0,Y 480.872,Z 61.898,A -85,B 0,C 180,E1 23409.817,E2 23409.817} C_VEL
LIN {X 0,Y 480.894,Z 61.9,A -85,B 0,C 180,E1 23406.207,E2 23406.207} C_VEL
LIN {X 0,Y 480.871,Z 61.898,A -85,B 0,C 180,E1 23402.622,E2 23402.622} C_VEL
LIN {X 0,Y 480.842,Z 61.899,A -85,B 0,C 180,E1 23399.166,E2 23399.166} C_VEL
LIN {X 0,Y 480.838,Z 61.901,A -85,B 0,C 180,E1 23395.588,E2 23395.588} C_VEL
LIN {X 0,Y 480.859,Z 61.9,A -85,B 0,C 180,E1 23392.112,E2 23392.112} C_VEL
LIN {X 0,Y 480.886,Z 61.899,A -85,B 0,C 180,E1 23388.608,E2 23388.608} C_VEL
LIN {X 0,Y 480.855,Z 61.898,A -85,B 0,C 180,E1 23385.058,E2 23385.058} C_VEL
LIN {X 0,Y 480.831,Z 61.898,A -85,B 0,C 180,E1 23381.575,E2 23381.575} C_VEL
LIN {X 0,Y 480.83,Z 61.901,A -85,B 0,C 180,E1 23378.019,E2 23378.019} C_VEL
LIN {X 0,Y 480.867,Z 61.901,A -85,B 0,C 180,E1 23374.638,E2 23374.638} C_VEL
LIN {X 0,Y 480.879,Z 61.898,A -85,B 0,C 180,E1 23371.023,E2 23371.023} C_VEL
LIN {X 0,Y 480.837,Z 61.902,A -85,B 0,C 180,E1 23367.555,E2 23367.555} C_VEL
LIN {X 0,Y 480.82,Z 61.902,A -85,B 0,C 180,E1 23364.097,E2 23364.097} C_VEL
LIN {X 0,Y 480.835,Z 61.904,A -85,B 0,C 180,E1 23360.638,E2 23360.638} C_VEL
LIN {X 0,Y 480.869,Z 61.902,A -85,B 0,C 180,E1 23357.163,E2 23357.163} C_VEL
LIN {X 0,Y 480.848,Z 61.899,A -85,B 0,C 180,E1 23353.646,E2 23353.646} C_VEL
LIN {X 0,Y 480.821,Z 61.906,A -85,B 0,C 180,E1 23350.256,E2 23350.256} C_VEL
LIN {X 0,Y 480.864,Z 62.122,A -85,B 0,C 180,E1 23346.829,E2 23346.829} C_VEL
LIN {X 0,Y 486.36,Z 77.333,A -85,B 0,C 180,E1 23344.786,E2 23344.786} C_VEL
LIN {X 0,Y 490.758,Z 91.081,A -85,B 0,C 180,E1 23343.138,E2 23343.138} C_VEL
LIN {X 0,Y 487.97,Z 134.217,A -85,B 0,C 180,E1 23339.39,E2 23339.39} C_VEL
LIN {X 0,Y 486.704,Z 160.033,A -85,B 0,C 180,E1 23337.245,E2 23337.245} C_VEL
LIN {X 0,Y 488.353,Z 175.465,A -85,B 0,C 180,E1 23336.92,E2 23336.92} C_VEL
LIN {X 0,Y 486.768,Z 361.485,A -85,B 0,C 180,E1 23334.148,E2 23334.148} C_VEL
LIN {X 0,Y 486.201,Z 380.198,A -85,B 0,C 180,E1 23333.658,E2 23333.658} C_VEL
LIN {X 0,Y 485.502,Z 397.721,A -85,B 0,C 180,E1 23332.991,E2 23332.991} C_VEL
LIN {X 0,Y 484.679,Z 415.013,A -85,B 0,C 180,E1 23332.117,E2 23332.117} C_VEL
LIN {X 0,Y 483.8,Z 432.163,A -85,B 0,C 180,E1 23331.013,E2 23331.013} C_VEL
LIN {X 0,Y 482.936,Z 448.366,A -85,B 0,C 180,E1 23329.723,E2 23329.723} C_VEL
LIN {X 0,Y 482.124,Z 463.816,A -85,B 0,C 180,E1 23328.227,E2 23328.227} C_VEL
LIN {X 0,Y 481.467,Z 477.321,A -85,B 0,C 180,E1 23326.654,E2 23326.654} C_VEL
LIN {X 0,Y 480.9,Z 490.47,A -85,B 0,C 180,E1 23324.818,E2 23324.818} C_VEL
LIN {X 0,Y 480.541,Z 501.325,A -85,B 0,C 180,E1 23322.987,E2 23322.987} C_VEL
LIN {X 0,Y 480.308,Z 510.82,A -85,B 0,C 180,E1 23321.042,E2 23321.042} C_VEL
LIN {X 0,Y 480.22,Z 518.893,A -85,B 0,C 180,E1 23318.985,E2 23318.985} C_VEL
LIN {X 0,Y 480.206,Z 525.108,A -85,B 0,C 180,E1 23316.937,E2 23316.937} C_VEL
LIN {X 0,Y 480.238,Z 529.846,A -85,B 0,C 180,E1 23314.778,E2 23314.778} C_VEL
LIN {X 0,Y 480.277,Z 532.802,A -85,B 0,C 180,E1 23312.626,E2 23312.626} C_VEL
LIN {X 0,Y 480.298,Z 534.05,A -85,B 0,C 180,E1 23310.478,E2 23310.478} C_VEL
LIN {X 0,Y 480.286,Z 533.612,A -85,B 0,C 180,E1 23308.331,E2 23308.331} C_VEL
LIN {X 0,Y 480.242,Z 531.483,A -85,B 0,C 180,E1 23306.181,E2 23306.181} C_VEL
LIN {X 0,Y 480.199,Z 527.614,A -85,B 0,C 180,E1 23304.025,E2 23304.025} C_VEL
LIN {X 0,Y 480.185,Z 521.913,A -85,B 0,C 180,E1 23301.861,E2 23301.861} C_VEL
LIN {X 0,Y 480.244,Z 514.238,A -85,B 0,C 180,E1 23299.687,E2 23299.687} C_VEL
LIN {X 0,Y 480.444,Z 504.962,A -85,B 0,C 180,E1 23297.623,E2 23297.623} C_VEL
LIN {X 0,Y 480.797,Z 494.142,A -85,B 0,C 180,E1 23295.673,E2 23295.673} C_VEL
LIN {X 0,Y 481.32,Z 481.806,A -85,B 0,C 180,E1 23293.839,E2 23293.839} C_VEL
LIN {X 0,Y 482.009,Z 467.892,A -85,B 0,C 180,E1 23292.122,E2 23292.122} C_VEL
LIN {X 0,Y 482.819,Z 452.835,A -85,B 0,C 180,E1 23290.588,E2 23290.588} C_VEL
LIN {X 0,Y 483.718,Z 436.557,A -85,B 0,C 180,E1 23289.228,E2 23289.228} C_VEL
LIN {X 0,Y 484.571,Z 420.543,A -85,B 0,C 180,E1 23288.135,E2 23288.135} C_VEL
LIN {X 0,Y 485.39,Z 403.741,A -85,B 0,C 180,E1 23287.217,E2 23287.217} C_VEL
LIN {X 0,Y 486.159,Z 385.597,A -85,B 0,C 180,E1 23286.462,E2 23286.462} C_VEL
LIN {X 0,Y 486.793,Z 366.963,A -85,B 0,C 180,E1 23285.918,E2 23285.918} C_VEL
LIN {X 0,Y 487.135,Z 344.345,A -85,B 0,C 180,E1 23285.52,E2 23285.52} C_VEL
LIN {X 0,Y 488.492,Z 164.563,A -85,B 0,C 180,E1 23282.849,E2 23282.849} C_VEL
LIN {X 0,Y 487.999,Z 155.292,A -85,B 0,C 180,E1 23282.649,E2 23282.649} C_VEL
LIN {X 0,Y 490.516,Z 86.839,A -85,B 0,C 180,E1 23279.253,E2 23279.253} C_VEL
LIN {X 0,Y 480.962,Z 62.395,A -85,B 0,C 180,E1 23277.319,E2 23277.319} C_VEL
LIN {X 0,Y 480.881,Z 61.909,A -85,B 0,C 180,E1 23277.136,E2 23277.136} C_VEL
LIN {X 0,Y 480.885,Z 61.897,A -85,B 0,C 180,E1 23273.514,E2 23273.514} C_VEL
LIN {X 0,Y 480.891,Z 61.896,A -85,B 0,C 180,E1 23269.87,E2 23269.87} C_VEL
LIN {X 0,Y 480.888,Z 61.897,A -85,B 0,C 180,E1 23266.184,E2 23266.184} C_VEL
LIN {X 0,Y 480.888,Z 61.895,A -85,B 0,C 180,E1 23262.511,E2 23262.511} C_VEL
LIN {X 0,Y 480.892,Z 61.892,A -85,B 0,C 180,E1 23258.896,E2 23258.896} C_VEL
LIN {X 0,Y 480.876,Z 61.891,A -85,B 0,C 180,E1 23255.312,E2 23255.312} C_VEL
LIN {X 0,Y 480.874,Z 61.894,A -85,B 0,C 180,E1 23251.739,E2 23251.739} C_VEL
LIN {X 0,Y 480.888,Z 61.893,A -85,B 0,C 180,E1 23248.163,E2 23248.163} C_VEL
LIN {X 0,Y 480.891,Z 61.897,A -85,B 0,C 180,E1 23244.572,E2 23244.572} C_VEL
LIN {X 0,Y 480.894,Z 61.894,A -85,B 0,C 180,E1 23240.954,E2 23240.954} C_VEL
LIN {X 0,Y 480.884,Z 61.892,A -85,B 0,C 180,E1 23237.297,E2 23237.297} C_VEL
LIN {X 0,Y 480.867,Z 61.891,A -85,B 0,C 180,E1 23233.712,E2 23233.712} C_VEL
LIN {X 0,Y 480.863,Z 61.89,A -85,B 0,C 180,E1 23230.059,E2 23230.059} C_VEL
LIN {X 0,Y 480.872,Z 61.896,A -85,B 0,C 180,E1 23226.447,E2 23226.447} C_VEL
LIN {X 0,Y 480.887,Z 61.897,A -85,B 0,C 180,E1 23222.86,E2 23222.86} C_VEL
LIN {X 0,Y 480.897,Z 61.888,A -85,B 0,C 180,E1 23219.285,E2 23219.285} C_VEL
LIN {X 0,Y 480.88,Z 61.892,A -85,B 0,C 180,E1 23215.707,E2 23215.707} C_VEL
LIN {X 0,Y 480.857,Z 61.896,A -85,B 0,C 180,E1 23212.232,E2 23212.232} C_VEL
LIN {X 0,Y 480.856,Z 61.898,A -85,B 0,C 180,E1 23208.607,E2 23208.607} C_VEL
LIN {X 0,Y 480.875,Z 61.899,A -85,B 0,C 180,E1 23205.059,E2 23205.059} C_VEL
LIN {X 0,Y 480.892,Z 61.893,A -85,B 0,C 180,E1 23201.451,E2 23201.451} C_VEL
LIN {X 0,Y 480.898,Z 61.887,A -85,B 0,C 180,E1 23197.765,E2 23197.765} C_VEL
LIN {X 0,Y 480.874,Z 61.891,A -85,B 0,C 180,E1 23194.11,E2 23194.11} C_VEL
LIN {X 0,Y 480.848,Z 61.889,A -85,B 0,C 180,E1 23190.601,E2 23190.601} C_VEL
LIN {X 0,Y 480.846,Z 61.9,A -85,B 0,C 180,E1 23186.989,E2 23186.989} C_VEL
LIN {X 0,Y 480.865,Z 61.894,A -85,B 0,C 180,E1 23183.51,E2 23183.51} C_VEL
LIN {X 0,Y 480.894,Z 61.89,A -85,B 0,C 180,E1 23180.024,E2 23180.024} C_VEL
LIN {X 0,Y 480.863,Z 61.896,A -85,B 0,C 180,E1 23176.508,E2 23176.508} C_VEL
LIN {X 0,Y 480.84,Z 61.894,A -85,B 0,C 180,E1 23173.001,E2 23173.001} C_VEL
LIN {X 0,Y 480.836,Z 61.904,A -85,B 0,C 180,E1 23169.326,E2 23169.326} C_VEL
LIN {X 0,Y 480.91,Z 62.101,A -85,B 0,C 180,E1 23166.148,E2 23166.148} C_VEL
LIN {X 0,Y 484.885,Z 77.9,A -85,B 0,C 180,E1 23164.219,E2 23164.219} C_VEL
LIN {X 0,Y 484.677,Z 110.333,A -85,B 0,C 180,E1 23160.717,E2 23160.717} C_VEL
LIN {X 0,Y 484.662,Z 111.429,A -85,B 0,C 180,E1 23160.597,E2 23160.597} C_VEL
LIN {X 0,Y 483.666,Z 117.304,A -85,B 0,C 180,E1 23160.008,E2 23160.008} C_VEL
LIN {X 0,Y 477.36,Z 134.434,A -85,B 0,C 180,E1 23158.462,E2 23158.462} C_VEL
LIN {X 0,Y 476.791,Z 138.63,A -85,B 0,C 180,E1 23158.028,E2 23158.028} C_VEL
LIN {X 0,Y 476.364,Z 172.456,A -85,B 0,C 180,E1 23154.363,E2 23154.363} C_VEL
LIN {X 0,Y 476.367,Z 187.713,A -85,B 0,C 180,E1 23152.795,E2 23152.795} C_VEL
LIN {X 0,Y 476.853,Z 192.942,A -85,B 0,C 180,E1 23152.69,E2 23152.69} C_VEL
LIN {X 0,Y 476.063,Z 299.297,A -85,B 0,C 180,E1 23151.038,E2 23151.038} C_VEL
LIN {X 0,Y 476,Z 313.737,A -85,B 0,C 180,E1 23150.601,E2 23150.601} C_VEL
LIN {X 0,Y 475.766,Z 327.51,A -85,B 0,C 180,E1 23149.967,E2 23149.967} C_VEL
LIN {X 0,Y 475.349,Z 341.155,A -85,B 0,C 180,E1 23149.09,E2 23149.09} C_VEL
LIN {X 0,Y 474.904,Z 352.917,A -85,B 0,C 180,E1 23148.096,E2 23148.096} C_VEL
LIN {X 0,Y 474.435,Z 364.008,A -85,B 0,C 180,E1 23146.903,E2 23146.903} C_VEL
LIN {X 0,Y 473.906,Z 374.718,A -85,B 0,C 180,E1 23145.416,E2 23145.416} C_VEL
LIN {X 0,Y 473.455,Z 383.575,A -85,B 0,C 180,E1 23143.805,E2 23143.805} C_VEL
LIN {X 0,Y 473.125,Z 390.229,A -85,B 0,C 180,E1 23142.199,E2 23142.199} C_VEL
LIN {X 0,Y 472.894,Z 395.398,A -85,B 0,C 180,E1 23140.475,E2 23140.475} C_VEL
LIN {X 0,Y 472.735,Z 398.943,A -85,B 0,C 180,E1 23138.636,E2 23138.636} C_VEL
LIN {X 0,Y 472.658,Z 400.65,A -85,B 0,C 180,E1 23136.68,E2 23136.68} C_VEL
LIN {X 0,Y 472.657,Z 400.317,A -85,B 0,C 180,E1 23134.731,E2 23134.731} C_VEL
LIN {X 0,Y 472.724,Z 398.158,A -85,B 0,C 180,E1 23132.909,E2 23132.909} C_VEL
LIN {X 0,Y 472.866,Z 394.487,A -85,B 0,C 180,E1 23131.211,E2 23131.211} C_VEL
LIN {X 0,Y 473.087,Z 389.034,A -85,B 0,C 180,E1 23129.515,E2 23129.515} C_VEL
LIN {X 0,Y 473.418,Z 381.483,A -85,B 0,C 180,E1 23127.82,E2 23127.82} C_VEL
LIN {X 0,Y 473.807,Z 372.986,A -85,B 0,C 180,E1 23126.369,E2 23126.369} C_VEL
LIN {X 0,Y 474.251,Z 363.092,A -85,B 0,C 180,E1 23125.04,E2 23125.04} C_VEL
LIN {X 0,Y 474.715,Z 351.039,A -85,B 0,C 180,E1 23123.778,E2 23123.778} C_VEL
LIN {X 0,Y 475.151,Z 338.136,A -85,B 0,C 180,E1 23122.746,E2 23122.746} C_VEL
LIN {X 0,Y 475.489,Z 325.098,A -85,B 0,C 180,E1 23121.961,E2 23121.961} C_VEL
LIN {X 0,Y 475.656,Z 310.759,A -85,B 0,C 180,E1 23121.34,E2 23121.34} C_VEL
LIN {X 0,Y 475.687,Z 295.263,A -85,B 0,C 180,E1 23120.925,E2 23120.925} C_VEL
LIN {X 0,Y 476.562,Z 183.387,A -85,B 0,C 180,E1 23119.207,E2 23119.207} C_VEL
LIN {X 0,Y 477.107,Z 131.301,A -85,B 0,C 180,E1 23115.868,E2 23115.868} C_VEL
LIN {X 0,Y 477.595,Z 97.253,A -85,B 0,C 180,E1 23113.614,E2 23113.614} C_VEL
LIN {X 0,Y 478.025,Z 96.2,A -85,B 0,C 180,E1 23113.41,E2 23113.41} C_VEL
LIN {X 0,Y 479.843,Z 97.111,A -85,B 0,C 180,E1 23113.148,E2 23113.148} C_VEL
LIN {X 0,Y 477.917,Z 144.958,A -85,B 0,C 180,E1 23109.55,E2 23109.55} C_VEL
LIN {X 0,Y 477.021,Z 171.535,A -85,B 0,C 180,E1 23107.594,E2 23107.594} C_VEL
LIN {X 0,Y 478.347,Z 186.167,A -85,B 0,C 180,E1 23107.285,E2 23107.285} C_VEL
LIN {X 0,Y 476.942,Z 293.69,A -85,B 0,C 180,E1 23105.49,E2 23105.49} C_VEL
LIN {X 0,Y 476.669,Z 308.668,A -85,B 0,C 180,E1 23105.026,E2 23105.026} C_VEL
LIN {X 0,Y 476.247,Z 322.748,A -85,B 0,C 180,E1 23104.374,E2 23104.374} C_VEL
LIN {X 0,Y 475.699,Z 336.86,A -85,B 0,C 180,E1 23103.488,E2 23103.488} C_VEL
LIN {X 0,Y 475.082,Z 350.237,A -85,B 0,C 180,E1 23102.38,E2 23102.38} C_VEL
LIN {X 0,Y 474.49,Z 362.162,A -85,B 0,C 180,E1 23101.105,E2 23101.105} C_VEL
LIN {X 0,Y 473.955,Z 372.405,A -85,B 0,C 180,E1 23099.722,E2 23099.722} C_VEL
LIN {X 0,Y 473.471,Z 381.789,A -85,B 0,C 180,E1 23098.096,E2 23098.096} C_VEL
LIN {X 0,Y 473.106,Z 389.259,A -85,B 0,C 180,E1 23096.375,E2 23096.375} C_VEL
LIN {X 0,Y 472.881,Z 394.588,A -85,B 0,C 180,E1 23094.703,E2 23094.703} C_VEL
LIN {X 0,Y 472.738,Z 398.486,A -85,B 0,C 180,E1 23092.88,E2 23092.88} C_VEL
LIN {X 0,Y 472.671,Z 400.508,A -85,B 0,C 180,E1 23091.078,E2 23091.078} C_VEL
LIN {X 0,Y 472.688,Z 400.84,A -85,B 0,C 180,E1 23089.185,E2 23089.185} C_VEL
LIN {X 0,Y 472.783,Z 399.163,A -85,B 0,C 180,E1 23087.211,E2 23087.211} C_VEL
LIN {X 0,Y 472.954,Z 395.789,A -85,B 0,C 180,E1 23085.422,E2 23085.422} C_VEL
LIN {X 0,Y 473.221,Z 390.812,A -85,B 0,C 180,E1 23083.703,E2 23083.703} C_VEL
LIN {X 0,Y 473.634,Z 383.456,A -85,B 0,C 180,E1 23081.908,E2 23081.908} C_VEL
LIN {X 0,Y 474.132,Z 374.943,A -85,B 0,C 180,E1 23080.347,E2 23080.347} C_VEL
LIN {X 0,Y 474.697,Z 365.587,A -85,B 0,C 180,E1 23078.992,E2 23078.992} C_VEL
LIN {X 0,Y 475.332,Z 354.138,A -85,B 0,C 180,E1 23077.687,E2 23077.687} C_VEL
LIN {X 0,Y 475.989,Z 341.695,A -85,B 0,C 180,E1 23076.57,E2 23076.57} C_VEL
LIN {X 0,Y 476.624,Z 327.374,A -85,B 0,C 180,E1 23075.583,E2 23075.583} C_VEL
LIN {X 0,Y 477.126,Z 312.417,A -85,B 0,C 180,E1 23074.831,E2 23074.831} C_VEL
LIN {X 0,Y 477.467,Z 297.342,A -85,B 0,C 180,E1 23074.313,E2 23074.313} C_VEL
LIN {X 0,Y 477.848,Z 272.734,A -85,B 0,C 180,E1 23073.83,E2 23073.83} C_VEL
LIN {X 0,Y 479.064,Z 190.665,A -85,B 0,C 180,E1 23072.39,E2 23072.39} C_VEL
LIN {X 0,Y 476.048,Z 174.264,A -85,B 0,C 180,E1 23071.904,E2 23071.904} C_VEL
LIN {X 0,Y 477.512,Z 143.996,A -85,B 0,C 180,E1 23068.04,E2 23068.04} C_VEL
LIN {X 0,Y 479.246,Z 114.967,A -85,B 0,C 180,E1 23064.256,E2 23064.256} C_VEL
LIN {X 0,Y 480.846,Z 90.088,A -85,B 0,C 180,E1 23060.956,E2 23060.956} C_VEL
LIN {X 0,Y 476.23,Z 73.579,A -85,B 0,C 180,E1 23058.23,E2 23058.23} C_VEL
LIN {X 0,Y 472.956,Z 63.006,A -85,B 0,C 180,E1 23056.33,E2 23056.33} C_VEL
LIN {X 0,Y 472.912,Z 62.888,A -85,B 0,C 180,E1 23052.827,E2 23052.827} C_VEL
LIN {X 0,Y 472.905,Z 62.885,A -85,B 0,C 180,E1 23049.247,E2 23049.247} C_VEL
LIN {X 0,Y 472.917,Z 62.891,A -85,B 0,C 180,E1 23045.703,E2 23045.703} C_VEL
LIN {X 0,Y 472.947,Z 62.888,A -85,B 0,C 180,E1 23042.181,E2 23042.181} C_VEL
LIN {X 0,Y 472.935,Z 62.887,A -85,B 0,C 180,E1 23038.668,E2 23038.668} C_VEL
LIN {X 0,Y 472.905,Z 62.889,A -85,B 0,C 180,E1 23035.149,E2 23035.149} C_VEL
LIN {X 0,Y 472.896,Z 62.89,A -85,B 0,C 180,E1 23031.611,E2 23031.611} C_VEL
LIN {X 0,Y 472.907,Z 62.889,A -85,B 0,C 180,E1 23028.042,E2 23028.042} C_VEL
LIN {X 0,Y 472.943,Z 62.888,A -85,B 0,C 180,E1 23024.551,E2 23024.551} C_VEL
LIN {X 0,Y 472.937,Z 62.886,A -85,B 0,C 180,E1 23020.871,E2 23020.871} C_VEL
LIN {X 0,Y 472.903,Z 62.889,A -85,B 0,C 180,E1 23017.369,E2 23017.369} C_VEL
LIN {X 0,Y 472.888,Z 62.89,A -85,B 0,C 180,E1 23013.775,E2 23013.775} C_VEL
LIN {X 0,Y 472.886,Z 62.891,A -85,B 0,C 180,E1 23010.067,E2 23010.067} C_VEL
LIN {X 0,Y 472.908,Z 62.891,A -85,B 0,C 180,E1 23006.631,E2 23006.631} C_VEL
LIN {X 0,Y 472.933,Z 62.891,A -85,B 0,C 180,E1 23003.05,E2 23003.05} C_VEL
LIN {X 0,Y 472.907,Z 62.893,A -85,B 0,C 180,E1 22999.528,E2 22999.528} C_VEL
LIN {X 0,Y 472.881,Z 62.889,A -85,B 0,C 180,E1 22996.091,E2 22996.091} C_VEL
LIN {X 0,Y 472.882,Z 62.895,A -85,B 0,C 180,E1 22992.415,E2 22992.415} C_VEL
LIN {X 0,Y 472.9,Z 62.891,A -85,B 0,C 180,E1 22988.899,E2 22988.899} C_VEL
LIN {X 0,Y 472.969,Z 63.107,A -85,B 0,C 180,E1 22987.448,E2 22987.448} C_VEL
LIN {X 0,Y 478.697,Z 78.979,A -85,B 0,C 180,E1 22985.246,E2 22985.246} C_VEL
LIN {X 0,Y 483.524,Z 93.325,A -85,B 0,C 180,E1 22983.449,E2 22983.449} C_VEL
LIN {X 0,Y 480.434,Z 137.358,A -85,B 0,C 180,E1 22979.55,E2 22979.55} C_VEL
LIN {X 0,Y 479.219,Z 160.094,A -85,B 0,C 180,E1 22977.623,E2 22977.623} C_VEL
LIN {X 0,Y 480.953,Z 176.407,A -85,B 0,C 180,E1 22977.27,E2 22977.27} C_VEL
LIN {X 0,Y 479.249,Z 360.813,A -85,B 0,C 180,E1 22974.482,E2 22974.482} C_VEL
LIN {X 0,Y 478.645,Z 379.497,A -85,B 0,C 180,E1 22973.986,E2 22973.986} C_VEL
LIN {X 0,Y 477.86,Z 397.544,A -85,B 0,C 180,E1 22973.285,E2 22973.285} C_VEL
LIN {X 0,Y 476.95,Z 415.255,A -85,B 0,C 180,E1 22972.365,E2 22972.365} C_VEL
LIN {X 0,Y 475.967,Z 433.038,A -85,B 0,C 180,E1 22971.182,E2 22971.182} C_VEL
LIN {X 0,Y 475.053,Z 448.917,A -85,B 0,C 180,E1 22969.872,E2 22969.872} C_VEL
LIN {X 0,Y 474.23,Z 463.478,A -85,B 0,C 180,E1 22968.419,E2 22968.419} C_VEL
LIN {X 0,Y 473.505,Z 477.405,A -85,B 0,C 180,E1 22966.753,E2 22966.753} C_VEL
LIN {X 0,Y 472.93,Z 489.991,A -85,B 0,C 180,E1 22964.944,E2 22964.944} C_VEL
LIN {X 0,Y 472.537,Z 501.393,A -85,B 0,C 180,E1 22962.962,E2 22962.962} C_VEL
LIN {X 0,Y 472.305,Z 511.214,A -85,B 0,C 180,E1 22960.861,E2 22960.861} C_VEL
LIN {X 0,Y 472.237,Z 518.974,A -85,B 0,C 180,E1 22958.769,E2 22958.769} C_VEL
LIN {X 0,Y 472.243,Z 525.198,A -85,B 0,C 180,E1 22956.566,E2 22956.566} C_VEL
LIN {X 0,Y 472.299,Z 529.574,A -85,B 0,C 180,E1 22954.358,E2 22954.358} C_VEL
LIN {X 0,Y 472.355,Z 532.151,A -85,B 0,C 180,E1 22952.184,E2 22952.184} C_VEL
LIN {X 0,Y 472.381,Z 533.041,A -85,B 0,C 180,E1 22950.001,E2 22950.001} C_VEL
LIN {X 0,Y 472.346,Z 532.229,A -85,B 0,C 180,E1 22947.817,E2 22947.817} C_VEL
LIN {X 0,Y 472.28,Z 529.708,A -85,B 0,C 180,E1 22945.63,E2 22945.63} C_VEL
LIN {X 0,Y 472.221,Z 525.429,A -85,B 0,C 180,E1 22943.436,E2 22943.436} C_VEL
LIN {X 0,Y 472.215,Z 519.295,A -85,B 0,C 180,E1 22941.232,E2 22941.232} C_VEL
LIN {X 0,Y 472.289,Z 511.635,A -85,B 0,C 180,E1 22939.141,E2 22939.141} C_VEL
LIN {X 0,Y 472.533,Z 501.928,A -85,B 0,C 180,E1 22937.04,E2 22937.04} C_VEL
LIN {X 0,Y 472.943,Z 490.618,A -85,B 0,C 180,E1 22935.054,E2 22935.054} C_VEL
LIN {X 0,Y 473.512,Z 478.662,A -85,B 0,C 180,E1 22933.312,E2 22933.312} C_VEL
LIN {X 0,Y 474.258,Z 464.794,A -85,B 0,C 180,E1 22931.629,E2 22931.629} C_VEL
LIN {X 0,Y 475.115,Z 450.016,A -85,B 0,C 180,E1 22930.139,E2 22930.139} C_VEL
LIN {X 0,Y 476.05,Z 434.219,A -85,B 0,C 180,E1 22928.824,E2 22928.824} C_VEL
LIN {X 0,Y 477.042,Z 416.621,A -85,B 0,C 180,E1 22927.642,E2 22927.642} C_VEL
LIN {X 0,Y 477.964,Z 398.914,A -85,B 0,C 180,E1 22926.712,E2 22926.712} C_VEL
LIN {X 0,Y 478.754,Z 380.681,A -85,B 0,C 180,E1 22925.996,E2 22925.996} C_VEL
LIN {X 0,Y 479.362,Z 361.991,A -85,B 0,C 180,E1 22925.494,E2 22925.494} C_VEL
LIN {X 0,Y 479.885,Z 306.839,A -85,B 0,C 180,E1 22924.647,E2 22924.647} C_VEL
LIN {X 0,Y 481.051,Z 164.618,A -85,B 0,C 180,E1 22922.486,E2 22922.486} C_VEL
LIN {X 0,Y 480.569,Z 155.553,A -85,B 0,C 180,E1 22922.291,E2 22922.291} C_VEL
LIN {X 0,Y 483.189,Z 89.293,A -85,B 0,C 180,E1 22918.946,E2 22918.946} C_VEL
LIN {X 0,Y 473.044,Z 63.491,A -85,B 0,C 180,E1 22916.866,E2 22916.866} C_VEL
LIN {X 0,Y 472.951,Z 62.88,A -85,B 0,C 180,E1 22916.622,E2 22916.622} C_VEL
LIN {X 0,Y 472.943,Z 62.886,A -85,B 0,C 180,E1 22912.951,E2 22912.951} C_VEL
LIN {X 0,Y 472.943,Z 62.888,A -85,B 0,C 180,E1 22909.373,E2 22909.373} C_VEL
LIN {X 0,Y 472.949,Z 62.885,A -85,B 0,C 180,E1 22905.763,E2 22905.763} C_VEL
LIN {X 0,Y 472.954,Z 62.888,A -85,B 0,C 180,E1 22902.079,E2 22902.079} C_VEL
LIN {X 0,Y 472.95,Z 62.884,A -85,B 0,C 180,E1 22898.429,E2 22898.429} C_VEL
LIN {X 0,Y 472.953,Z 62.878,A -85,B 0,C 180,E1 22894.806,E2 22894.806} C_VEL
LIN {X 0,Y 472.947,Z 62.879,A -85,B 0,C 180,E1 22891.11,E2 22891.11} C_VEL
LIN {X 0,Y 472.932,Z 62.881,A -85,B 0,C 180,E1 22887.581,E2 22887.581} C_VEL
LIN {X 0,Y 472.933,Z 62.88,A -85,B 0,C 180,E1 22883.949,E2 22883.949} C_VEL
LIN {X 0,Y 472.949,Z 62.885,A -85,B 0,C 180,E1 22880.415,E2 22880.415} C_VEL
LIN {X 0,Y 472.955,Z 62.886,A -85,B 0,C 180,E1 22876.709,E2 22876.709} C_VEL
LIN {X 0,Y 472.955,Z 62.879,A -85,B 0,C 180,E1 22873.074,E2 22873.074} C_VEL
LIN {X 0,Y 472.941,Z 62.876,A -85,B 0,C 180,E1 22869.491,E2 22869.491} C_VEL
LIN {X 0,Y 472.923,Z 62.882,A -85,B 0,C 180,E1 22865.946,E2 22865.946} C_VEL
LIN {X 0,Y 472.923,Z 62.886,A -85,B 0,C 180,E1 22862.302,E2 22862.302} C_VEL
LIN {X 0,Y 472.94,Z 62.885,A -85,B 0,C 180,E1 22858.788,E2 22858.788} C_VEL
LIN {X 0,Y 472.951,Z 62.881,A -85,B 0,C 180,E1 22855.149,E2 22855.149} C_VEL
LIN {X 0,Y 472.957,Z 62.884,A -85,B 0,C 180,E1 22851.49,E2 22851.49} C_VEL
LIN {X 0,Y 472.942,Z 62.884,A -85,B 0,C 180,E1 22847.795,E2 22847.795} C_VEL
LIN {X 0,Y 472.917,Z 62.885,A -85,B 0,C 180,E1 22844.298,E2 22844.298} C_VEL
LIN {X 0,Y 472.913,Z 62.886,A -85,B 0,C 180,E1 22840.613,E2 22840.613} C_VEL
LIN {X 0,Y 472.916,Z 62.867,A -85,B 0,C 180,E1 22836.975,E2 22836.975} C_VEL
LIN {X 0,Y 472.937,Z 62.889,A -85,B 0,C 180,E1 22833.371,E2 22833.371} C_VEL
LIN {X 0,Y 472.96,Z 62.869,A -85,B 0,C 180,E1 22829.791,E2 22829.791} C_VEL
LIN {X 0,Y 472.949,Z 62.887,A -85,B 0,C 180,E1 22826.074,E2 22826.074} C_VEL
LIN {X 0,Y 472.923,Z 62.887,A -85,B 0,C 180,E1 22822.448,E2 22822.448} C_VEL
LIN {X 0,Y 472.905,Z 62.886,A -85,B 0,C 180,E1 22818.887,E2 22818.887} C_VEL
LIN {X 0,Y 472.901,Z 62.89,A -85,B 0,C 180,E1 22815.245,E2 22815.245} C_VEL
LIN {X 0,Y 472.921,Z 62.892,A -85,B 0,C 180,E1 22811.727,E2 22811.727} C_VEL
LIN {X 0,Y 472.95,Z 62.883,A -85,B 0,C 180,E1 22808.145,E2 22808.145} C_VEL
LIN {X 0,Y 472.977,Z 63.183,A -85,B 0,C 180,E1 22806.495,E2 22806.495} C_VEL
LIN {X 0,Y 477.335,Z 79.889,A -85,B 0,C 180,E1 22804.439,E2 22804.439} C_VEL
LIN {X 0,Y 477.119,Z 111.532,A -85,B 0,C 180,E1 22801.006,E2 22801.006} C_VEL
LIN {X 0,Y 476.791,Z 138.63,A -85,B 0,C 180,E1 22798.028,E2 22798.028} C_VEL
LIN {X 0,Y 475.774,Z 144.542,A -85,B 0,C 180,E1 22797.436,E2 22797.436} C_VEL
LIN {X 0,Y 469.685,Z 160.987,A -85,B 0,C 180,E1 22795.976,E2 22795.976} C_VEL
LIN {X 0,Y 468.92,Z 166.096,A -85,B 0,C 180,E1 22795.46,E2 22795.46} C_VEL
LIN {X 0,Y 468.796,Z 188.702,A -85,B 0,C 180,E1 22793.102,E2 22793.102} C_VEL
LIN {X 0,Y 469.288,Z 193.958,A -85,B 0,C 180,E1 22792.995,E2 22792.995} C_VEL
LIN {X 0,Y 468.441,Z 300.277,A -85,B 0,C 180,E1 22791.315,E2 22791.315} C_VEL
LIN {X 0,Y 468.375,Z 314.749,A -85,B 0,C 180,E1 22790.872,E2 22790.872} C_VEL
LIN {X 0,Y 468.131,Z 328.274,A -85,B 0,C 180,E1 22790.242,E2 22790.242} C_VEL
LIN {X 0,Y 467.687,Z 342.01,A -85,B 0,C 180,E1 22789.351,E2 22789.351} C_VEL
LIN {X 0,Y 467.207,Z 353.887,A -85,B 0,C 180,E1 22788.335,E2 22788.335} C_VEL
LIN {X 0,Y 466.674,Z 365.43,A -85,B 0,C 180,E1 22787.068,E2 22787.068} C_VEL
LIN {X 0,Y 466.122,Z 375.77,A -85,B 0,C 180,E1 22785.605,E2 22785.605} C_VEL
LIN {X 0,Y 465.617,Z 384.859,A -85,B 0,C 180,E1 22783.922,E2 22783.922} C_VEL
LIN {X 0,Y 465.234,Z 391.924,A -85,B 0,C 180,E1 22782.157,E2 22782.157} C_VEL
LIN {X 0,Y 464.98,Z 396.887,A -85,B 0,C 180,E1 22780.405,E2 22780.405} C_VEL
LIN {X 0,Y 464.82,Z 400.093,A -85,B 0,C 180,E1 22778.659,E2 22778.659} C_VEL
LIN {X 0,Y 464.734,Z 401.758,A -85,B 0,C 180,E1 22776.671,E2 22776.671} C_VEL
LIN {X 0,Y 464.733,Z 401.386,A -85,B 0,C 180,E1 22774.688,E2 22774.688} C_VEL
LIN {X 0,Y 464.815,Z 398.981,A -85,B 0,C 180,E1 22772.711,E2 22772.711} C_VEL
LIN {X 0,Y 464.989,Z 394.744,A -85,B 0,C 180,E1 22770.847,E2 22770.847} C_VEL
LIN {X 0,Y 465.243,Z 388.986,A -85,B 0,C 180,E1 22769.137,E2 22769.137} C_VEL
LIN {X 0,Y 465.593,Z 381.724,A -85,B 0,C 180,E1 22767.538,E2 22767.538} C_VEL
LIN {X 0,Y 466.062,Z 372.166,A -85,B 0,C 180,E1 22765.939,E2 22765.939} C_VEL
LIN {X 0,Y 466.572,Z 361.164,A -85,B 0,C 180,E1 22764.527,E2 22764.527} C_VEL
LIN {X 0,Y 467.02,Z 349.483,A -85,B 0,C 180,E1 22763.36,E2 22763.36} C_VEL
LIN {X 0,Y 467.441,Z 337.696,A -85,B 0,C 180,E1 22762.44,E2 22762.44} C_VEL
LIN {X 0,Y 467.785,Z 324.109,A -85,B 0,C 180,E1 22761.642,E2 22761.642} C_VEL
LIN {X 0,Y 467.933,Z 309.641,A -85,B 0,C 180,E1 22761.045,E2 22761.045} C_VEL
LIN {X 0,Y 467.941,Z 294.851,A -85,B 0,C 180,E1 22760.671,E2 22760.671} C_VEL
LIN {X 0,Y 468.847,Z 184.656,A -85,B 0,C 180,E1 22758.965,E2 22758.965} C_VEL
LIN {X 0,Y 469.321,Z 140.376,A -85,B 0,C 180,E1 22756.132,E2 22756.132} C_VEL
LIN {X 0,Y 469.926,Z 102.577,A -85,B 0,C 180,E1 22753.625,E2 22753.625} C_VEL
LIN {X 0,Y 470.394,Z 101.618,A -85,B 0,C 180,E1 22753.419,E2 22753.419} C_VEL
LIN {X 0,Y 472.262,Z 102.878,A -85,B 0,C 180,E1 22753.131,E2 22753.131} C_VEL
LIN {X 0,Y 470.022,Z 155.542,A -85,B 0,C 180,E1 22749.125,E2 22749.125} C_VEL
LIN {X 0,Y 469.474,Z 171.529,A -85,B 0,C 180,E1 22747.952,E2 22747.952} C_VEL
LIN {X 0,Y 470.861,Z 187.082,A -85,B 0,C 180,E1 22747.616,E2 22747.616} C_VEL
LIN {X 0,Y 469.357,Z 294.289,A -85,B 0,C 180,E1 22745.79,E2 22745.79} C_VEL
LIN {X 0,Y 469.057,Z 309.637,A -85,B 0,C 180,E1 22745.304,E2 22745.304} C_VEL
LIN {X 0,Y 468.581,Z 324.335,A -85,B 0,C 180,E1 22744.602,E2 22744.602} C_VEL
LIN {X 0,Y 468.031,Z 337.539,A -85,B 0,C 180,E1 22743.754,E2 22743.754} C_VEL
LIN {X 0,Y 467.359,Z 351.216,A -85,B 0,C 180,E1 22742.604,E2 22742.604} C_VEL
LIN {X 0,Y 466.732,Z 363.014,A -85,B 0,C 180,E1 22741.323,E2 22741.323} C_VEL
LIN {X 0,Y 466.159,Z 373.225,A -85,B 0,C 180,E1 22739.926,E2 22739.926} C_VEL
LIN {X 0,Y 465.626,Z 382.776,A -85,B 0,C 180,E1 22738.25,E2 22738.25} C_VEL
LIN {X 0,Y 465.224,Z 390.381,A -85,B 0,C 180,E1 22736.472,E2 22736.472} C_VEL
LIN {X 0,Y 464.98,Z 395.625,A -85,B 0,C 180,E1 22734.799,E2 22734.799} C_VEL
LIN {X 0,Y 464.823,Z 399.551,A -85,B 0,C 180,E1 22732.944,E2 22732.944} C_VEL
LIN {X 0,Y 464.749,Z 401.622,A -85,B 0,C 180,E1 22731.082,E2 22731.082} C_VEL
LIN {X 0,Y 464.766,Z 401.983,A -85,B 0,C 180,E1 22729.224,E2 22729.224} C_VEL
LIN {X 0,Y 464.855,Z 400.525,A -85,B 0,C 180,E1 22727.348,E2 22727.348} C_VEL
LIN {X 0,Y 465.046,Z 397.321,A -85,B 0,C 180,E1 22725.5,E2 22725.5} C_VEL
LIN {X 0,Y 465.355,Z 392.044,A -85,B 0,C 180,E1 22723.607,E2 22723.607} C_VEL
LIN {X 0,Y 465.783,Z 385.052,A -85,B 0,C 180,E1 22721.851,E2 22721.851} C_VEL
LIN {X 0,Y 466.285,Z 377.3,A -85,B 0,C 180,E1 22720.36,E2 22720.36} C_VEL
LIN {X 0,Y 466.963,Z 366.831,A -85,B 0,C 180,E1 22718.795,E2 22718.795} C_VEL
LIN {X 0,Y 467.663,Z 355.257,A -85,B 0,C 180,E1 22717.446,E2 22717.446} C_VEL
LIN {X 0,Y 468.347,Z 343.368,A -85,B 0,C 180,E1 22716.349,E2 22716.349} C_VEL
LIN {X 0,Y 469.03,Z 329.081,A -85,B 0,C 180,E1 22715.334,E2 22715.334} C_VEL
LIN {X 0,Y 469.568,Z 314.603,A -85,B 0,C 180,E1 22714.574,E2 22714.574} C_VEL
LIN {X 0,Y 469.962,Z 299.355,A -85,B 0,C 180,E1 22714.016,E2 22714.016} C_VEL
LIN {X 0,Y 470.293,Z 278.616,A -85,B 0,C 180,E1 22713.581,E2 22713.581} C_VEL
LIN {X 0,Y 471.714,Z 191.774,A -85,B 0,C 180,E1 22712.018,E2 22712.018} C_VEL
LIN {X 0,Y 468.467,Z 173.997,A -85,B 0,C 180,E1 22711.472,E2 22711.472} C_VEL
LIN {X 0,Y 470.045,Z 144.432,A -85,B 0,C 180,E1 22707.628,E2 22707.628} C_VEL
LIN {X 0,Y 471.861,Z 116.036,A -85,B 0,C 180,E1 22703.874,E2 22703.874} C_VEL
LIN {X 0,Y 473.497,Z 93.015,A -85,B 0,C 180,E1 22700.779,E2 22700.779} C_VEL
LIN {X 0,Y 469.156,Z 77.236,A -85,B 0,C 180,E1 22698.129,E2 22698.129} C_VEL
LIN {X 0,Y 465.018,Z 64.014,A -85,B 0,C 180,E1 22695.719,E2 22695.719} C_VEL
LIN {X 0,Y 465.014,Z 63.877,A -85,B 0,C 180,E1 22692.165,E2 22692.165} C_VEL
LIN {X 0,Y 464.998,Z 63.871,A -85,B 0,C 180,E1 22688.463,E2 22688.463} C_VEL
LIN {X 0,Y 464.97,Z 63.879,A -85,B 0,C 180,E1 22684.935,E2 22684.935} C_VEL
LIN {X 0,Y 464.962,Z 63.877,A -85,B 0,C 180,E1 22681.356,E2 22681.356} C_VEL
LIN {X 0,Y 464.969,Z 63.878,A -85,B 0,C 180,E1 22677.782,E2 22677.782} C_VEL
LIN {X 0,Y 464.992,Z 63.876,A -85,B 0,C 180,E1 22674.2,E2 22674.2} C_VEL
LIN {X 0,Y 465.006,Z 63.877,A -85,B 0,C 180,E1 22670.595,E2 22670.595} C_VEL
LIN {X 0,Y 464.986,Z 63.877,A -85,B 0,C 180,E1 22666.927,E2 22666.927} C_VEL
LIN {X 0,Y 464.959,Z 63.875,A -85,B 0,C 180,E1 22663.381,E2 22663.381} C_VEL
LIN {X 0,Y 464.951,Z 63.877,A -85,B 0,C 180,E1 22659.744,E2 22659.744} C_VEL
LIN {X 0,Y 464.953,Z 63.879,A -85,B 0,C 180,E1 22656.056,E2 22656.056} C_VEL
LIN {X 0,Y 464.97,Z 63.88,A -85,B 0,C 180,E1 22652.463,E2 22652.463} C_VEL
LIN {X 0,Y 464.994,Z 63.877,A -85,B 0,C 180,E1 22648.849,E2 22648.849} C_VEL
LIN {X 0,Y 464.995,Z 63.877,A -85,B 0,C 180,E1 22645.113,E2 22645.113} C_VEL
LIN {X 0,Y 464.975,Z 63.88,A -85,B 0,C 180,E1 22641.421,E2 22641.421} C_VEL
LIN {X 0,Y 464.94,Z 63.883,A -85,B 0,C 180,E1 22638.025,E2 22638.025} C_VEL
LIN {X 0,Y 464.943,Z 63.883,A -85,B 0,C 180,E1 22634.34,E2 22634.34} C_VEL
LIN {X 0,Y 464.958,Z 63.879,A -85,B 0,C 180,E1 22630.804,E2 22630.804} C_VEL
LIN {X 0,Y 464.987,Z 64.133,A -85,B 0,C 180,E1 22628.093,E2 22628.093} C_VEL
LIN {X 0,Y 470.872,Z 80.036,A -85,B 0,C 180,E1 22625.792,E2 22625.792} C_VEL
LIN {X 0,Y 476.26,Z 96.051,A -85,B 0,C 180,E1 22623.731,E2 22623.731} C_VEL
LIN {X 0,Y 473.021,Z 138.999,A -85,B 0,C 180,E1 22619.855,E2 22619.855} C_VEL
LIN {X 0,Y 471.797,Z 160.429,A -85,B 0,C 180,E1 22618.011,E2 22618.011} C_VEL
LIN {X 0,Y 473.587,Z 177.224,A -85,B 0,C 180,E1 22617.636,E2 22617.636} C_VEL
LIN {X 0,Y 471.75,Z 360.21,A -85,B 0,C 180,E1 22614.826,E2 22614.826} C_VEL
LIN {X 0,Y 471.101,Z 378.885,A -85,B 0,C 180,E1 22614.323,E2 22614.323} C_VEL
LIN {X 0,Y 470.266,Z 396.729,A -85,B 0,C 180,E1 22613.621,E2 22613.621} C_VEL
LIN {X 0,Y 469.295,Z 414.496,A -85,B 0,C 180,E1 22612.683,E2 22612.683} C_VEL
LIN {X 0,Y 468.239,Z 432.245,A -85,B 0,C 180,E1 22611.483,E2 22611.483} C_VEL
LIN {X 0,Y 467.256,Z 448.092,A -85,B 0,C 180,E1 22610.153,E2 22610.153} C_VEL
LIN {X 0,Y 466.343,Z 463.156,A -85,B 0,C 180,E1 22608.619,E2 22608.619} C_VEL
LIN {X 0,Y 465.57,Z 477.014,A -85,B 0,C 180,E1 22606.918,E2 22606.918} C_VEL
LIN {X 0,Y 464.963,Z 489.464,A -85,B 0,C 180,E1 22605.083,E2 22605.083} C_VEL
LIN {X 0,Y 464.553,Z 500.798,A -85,B 0,C 180,E1 22603.062,E2 22603.062} C_VEL
LIN {X 0,Y 464.32,Z 510.499,A -85,B 0,C 180,E1 22600.924,E2 22600.924} C_VEL
LIN {X 0,Y 464.266,Z 518.177,A -85,B 0,C 180,E1 22598.796,E2 22598.796} C_VEL
LIN {X 0,Y 464.289,Z 524.049,A -85,B 0,C 180,E1 22596.679,E2 22596.679} C_VEL
LIN {X 0,Y 464.358,Z 528.427,A -85,B 0,C 180,E1 22594.447,E2 22594.447} C_VEL
LIN {X 0,Y 464.425,Z 531.038,A -85,B 0,C 180,E1 22592.222,E2 22592.222} C_VEL
LIN {X 0,Y 464.457,Z 531.937,A -85,B 0,C 180,E1 22590.001,E2 22590.001} C_VEL
LIN {X 0,Y 464.415,Z 531.126,A -85,B 0,C 180,E1 22587.78,E2 22587.78} C_VEL
LIN {X 0,Y 464.336,Z 528.589,A -85,B 0,C 180,E1 22585.546,E2 22585.546} C_VEL
LIN {X 0,Y 464.263,Z 524.311,A -85,B 0,C 180,E1 22583.323,E2 22583.323} C_VEL
LIN {X 0,Y 464.241,Z 518.154,A -85,B 0,C 180,E1 22581.08,E2 22581.08} C_VEL
LIN {X 0,Y 464.31,Z 510.464,A -85,B 0,C 180,E1 22578.952,E2 22578.952} C_VEL
LIN {X 0,Y 464.57,Z 500.709,A -85,B 0,C 180,E1 22576.814,E2 22576.814} C_VEL
LIN {X 0,Y 464.981,Z 490.049,A -85,B 0,C 180,E1 22574.905,E2 22574.905} C_VEL
LIN {X 0,Y 465.628,Z 477.329,A -85,B 0,C 180,E1 22573.021,E2 22573.021} C_VEL
LIN {X 0,Y 466.409,Z 463.813,A -85,B 0,C 180,E1 22571.357,E2 22571.357} C_VEL
LIN {X 0,Y 467.323,Z 449.112,A -85,B 0,C 180,E1 22569.852,E2 22569.852} C_VEL
LIN {X 0,Y 468.311,Z 433.454,A -85,B 0,C 180,E1 22568.529,E2 22568.529} C_VEL
LIN {X 0,Y 469.375,Z 415.749,A -85,B 0,C 180,E1 22567.323,E2 22567.323} C_VEL
LIN {X 0,Y 470.362,Z 397.906,A -85,B 0,C 180,E1 22566.375,E2 22566.375} C_VEL
LIN {X 0,Y 471.213,Z 379.598,A -85,B 0,C 180,E1 22565.65,E2 22565.65} C_VEL
LIN {X 0,Y 471.85,Z 360.957,A -85,B 0,C 180,E1 22565.148,E2 22565.148} C_VEL
LIN {X 0,Y 473.681,Z 165.879,A -85,B 0,C 180,E1 22562.142,E2 22562.142} C_VEL
LIN {X 0,Y 473.14,Z 155.653,A -85,B 0,C 180,E1 22561.921,E2 22561.921} C_VEL
LIN {X 0,Y 475.931,Z 91.927,A -85,B 0,C 180,E1 22558.649,E2 22558.649} C_VEL
LIN {X 0,Y 465.103,Z 64.438,A -85,B 0,C 180,E1 22556.372,E2 22556.372} C_VEL
LIN {X 0,Y 465.007,Z 63.867,A -85,B 0,C 180,E1 22556.096,E2 22556.096} C_VEL
LIN {X 0,Y 465.011,Z 63.875,A -85,B 0,C 180,E1 22552.365,E2 22552.365} C_VEL
LIN {X 0,Y 465.015,Z 63.873,A -85,B 0,C 180,E1 22548.695,E2 22548.695} C_VEL
LIN {X 0,Y 465.006,Z 63.873,A -85,B 0,C 180,E1 22544.977,E2 22544.977} C_VEL
LIN {X 0,Y 464.998,Z 63.871,A -85,B 0,C 180,E1 22541.309,E2 22541.309} C_VEL
LIN {X 0,Y 465,Z 63.876,A -85,B 0,C 180,E1 22537.638,E2 22537.638} C_VEL
LIN {X 0,Y 465.005,Z 63.877,A -85,B 0,C 180,E1 22533.906,E2 22533.906} C_VEL
LIN {X 0,Y 465.015,Z 63.876,A -85,B 0,C 180,E1 22530.193,E2 22530.193} C_VEL
LIN {X 0,Y 465.014,Z 63.871,A -85,B 0,C 180,E1 22526.564,E2 22526.564} C_VEL
LIN {X 0,Y 465.016,Z 63.865,A -85,B 0,C 180,E1 22522.903,E2 22522.903} C_VEL
LIN {X 0,Y 465.011,Z 63.866,A -85,B 0,C 180,E1 22519.207,E2 22519.207} C_VEL
LIN {X 0,Y 464.996,Z 63.871,A -85,B 0,C 180,E1 22515.575,E2 22515.575} C_VEL
LIN {X 0,Y 464.988,Z 63.874,A -85,B 0,C 180,E1 22511.913,E2 22511.913} C_VEL
LIN {X 0,Y 464.986,Z 63.874,A -85,B 0,C 180,E1 22508.159,E2 22508.159} C_VEL
LIN {X 0,Y 464.996,Z 63.87,A -85,B 0,C 180,E1 22504.563,E2 22504.563} C_VEL
LIN {X 0,Y 465.01,Z 63.87,A -85,B 0,C 180,E1 22500.862,E2 22500.862} C_VEL
LIN {X 0,Y 465.014,Z 63.875,A -85,B 0,C 180,E1 22497.165,E2 22497.165} C_VEL
LIN {X 0,Y 465.017,Z 63.87,A -85,B 0,C 180,E1 22493.456,E2 22493.456} C_VEL
LIN {X 0,Y 464.998,Z 63.867,A -85,B 0,C 180,E1 22489.844,E2 22489.844} C_VEL
LIN {X 0,Y 464.978,Z 63.868,A -85,B 0,C 180,E1 22486.317,E2 22486.317} C_VEL
LIN {X 0,Y 464.975,Z 63.871,A -85,B 0,C 180,E1 22482.608,E2 22482.608} C_VEL
LIN {X 0,Y 464.98,Z 63.872,A -85,B 0,C 180,E1 22478.941,E2 22478.941} C_VEL
LIN {X 0,Y 464.997,Z 63.859,A -85,B 0,C 180,E1 22475.345,E2 22475.345} C_VEL
LIN {X 0,Y 465.019,Z 63.872,A -85,B 0,C 180,E1 22471.768,E2 22471.768} C_VEL
LIN {X 0,Y 465.001,Z 63.868,A -85,B 0,C 180,E1 22468.137,E2 22468.137} C_VEL
LIN {X 0,Y 464.973,Z 63.866,A -85,B 0,C 180,E1 22464.583,E2 22464.583} C_VEL
LIN {X 0,Y 464.965,Z 63.876,A -85,B 0,C 180,E1 22460.944,E2 22460.944} C_VEL
LIN {X 0,Y 464.969,Z 63.877,A -85,B 0,C 180,E1 22457.341,E2 22457.341} C_VEL
LIN {X 0,Y 464.987,Z 63.873,A -85,B 0,C 180,E1 22453.738,E2 22453.738} C_VEL
LIN {X 0,Y 465.016,Z 63.87,A -85,B 0,C 180,E1 22450.167,E2 22450.167} C_VEL
LIN {X 0,Y 465.004,Z 64.141,A -85,B 0,C 180,E1 22446.896,E2 22446.896} C_VEL
LIN {X 0,Y 469.839,Z 82.322,A -85,B 0,C 180,E1 22444.623,E2 22444.623} C_VEL
LIN {X 0,Y 469.555,Z 114.374,A -85,B 0,C 180,E1 22441.128,E2 22441.128} C_VEL
LIN {X 0,Y 469.149,Z 146.907,A -85,B 0,C 180,E1 22437.545,E2 22437.545} C_VEL
LIN {X 0,Y 468.92,Z 166.096,A -85,B 0,C 180,E1 22435.46,E2 22435.46} C_VEL
LIN {X 0,Y 467.924,Z 170.167,A -85,B 0,C 180,E1 22435.078,E2 22435.078} C_VEL
LIN {X 0,Y 461.951,Z 181.386,A -85,B 0,C 180,E1 22434.223,E2 22434.223} C_VEL
LIN {X 0,Y 461.221,Z 184.922,A -85,B 0,C 180,E1 22433.891,E2 22433.891} C_VEL
LIN {X 0,Y 461.21,Z 189.49,A -85,B 0,C 180,E1 22433.426,E2 22433.426} C_VEL
LIN {X 0,Y 461.738,Z 194.779,A -85,B 0,C 180,E1 22433.312,E2 22433.312} C_VEL
LIN {X 0,Y 460.834,Z 300.973,A -85,B 0,C 180,E1 22431.61,E2 22431.61} C_VEL
LIN {X 0,Y 460.77,Z 315.436,A -85,B 0,C 180,E1 22431.166,E2 22431.166} C_VEL
LIN {X 0,Y 460.509,Z 329.066,A -85,B 0,C 180,E1 22430.526,E2 22430.526} C_VEL
LIN {X 0,Y 460.074,Z 342.027,A -85,B 0,C 180,E1 22429.684,E2 22429.684} C_VEL
LIN {X 0,Y 459.555,Z 354.179,A -85,B 0,C 180,E1 22428.651,E2 22428.651} C_VEL
LIN {X 0,Y 458.977,Z 365.899,A -85,B 0,C 180,E1 22427.363,E2 22427.363} C_VEL
LIN {X 0,Y 458.359,Z 376.549,A -85,B 0,C 180,E1 22425.846,E2 22425.846} C_VEL
LIN {X 0,Y 457.843,Z 384.99,A -85,B 0,C 180,E1 22424.285,E2 22424.285} C_VEL
LIN {X 0,Y 457.439,Z 391.861,A -85,B 0,C 180,E1 22422.624,E2 22422.624} C_VEL
LIN {X 0,Y 457.135,Z 397.219,A -85,B 0,C 180,E1 22420.841,E2 22420.841} C_VEL
LIN {X 0,Y 456.927,Z 400.899,A -85,B 0,C 180,E1 22418.937,E2 22418.937} C_VEL
LIN {X 0,Y 456.82,Z 402.698,A -85,B 0,C 180,E1 22417.039,E2 22417.039} C_VEL
LIN {X 0,Y 456.796,Z 402.724,A -85,B 0,C 180,E1 22415.148,E2 22415.148} C_VEL
LIN {X 0,Y 456.859,Z 400.988,A -85,B 0,C 180,E1 22413.261,E2 22413.261} C_VEL
LIN {X 0,Y 457.028,Z 397.09,A -85,B 0,C 180,E1 22411.253,E2 22411.253} C_VEL
LIN {X 0,Y 457.293,Z 391.33,A -85,B 0,C 180,E1 22409.373,E2 22409.373} C_VEL
LIN {X 0,Y 457.639,Z 384.423,A -85,B 0,C 180,E1 22407.745,E2 22407.745} C_VEL
LIN {X 0,Y 458.074,Z 376.169,A -85,B 0,C 180,E1 22406.245,E2 22406.245} C_VEL
LIN {X 0,Y 458.611,Z 365.524,A -85,B 0,C 180,E1 22404.745,E2 22404.745} C_VEL
LIN {X 0,Y 459.135,Z 353.459,A -85,B 0,C 180,E1 22403.434,E2 22403.434} C_VEL
LIN {X 0,Y 459.61,Z 340.704,A -85,B 0,C 180,E1 22402.373,E2 22402.373} C_VEL
LIN {X 0,Y 459.989,Z 327.812,A -85,B 0,C 180,E1 22401.562,E2 22401.562} C_VEL
LIN {X 0,Y 460.187,Z 313.262,A -85,B 0,C 180,E1 22400.903,E2 22400.903} C_VEL
LIN {X 0,Y 460.215,Z 297.562,A -85,B 0,C 180,E1 22400.466,E2 22400.466} C_VEL
LIN {X 0,Y 461.195,Z 185.305,A -85,B 0,C 180,E1 22398.684,E2 22398.684} C_VEL
LIN {X 0,Y 461.749,Z 138.004,A -85,B 0,C 180,E1 22395.644,E2 22395.644} C_VEL
LIN {X 0,Y 462.239,Z 107.903,A -85,B 0,C 180,E1 22393.635,E2 22393.635} C_VEL
LIN {X 0,Y 462.732,Z 107.063,A -85,B 0,C 180,E1 22393.427,E2 22393.427} C_VEL
LIN {X 0,Y 464.642,Z 108.299,A -85,B 0,C 180,E1 22393.143,E2 22393.143} C_VEL
LIN {X 0,Y 462.326,Z 160.047,A -85,B 0,C 180,E1 22389.159,E2 22389.159} C_VEL
LIN {X 0,Y 461.928,Z 171.364,A -85,B 0,C 180,E1 22388.326,E2 22388.326} C_VEL
LIN {X 0,Y 463.396,Z 187.778,A -85,B 0,C 180,E1 22387.963,E2 22387.963} C_VEL
LIN {X 0,Y 461.784,Z 294.802,A -85,B 0,C 180,E1 22386.101,E2 22386.101} C_VEL
LIN {X 0,Y 461.449,Z 310.678,A -85,B 0,C 180,E1 22385.586,E2 22385.586} C_VEL
LIN {X 0,Y 460.922,Z 325.902,A -85,B 0,C 180,E1 22384.838,E2 22384.838} C_VEL
LIN {X 0,Y 460.298,Z 339.562,A -85,B 0,C 180,E1 22383.924,E2 22383.924} C_VEL
LIN {X 0,Y 459.631,Z 352.371,A -85,B 0,C 180,E1 22382.817,E2 22382.817} C_VEL
LIN {X 0,Y 458.957,Z 364.212,A -85,B 0,C 180,E1 22381.503,E2 22381.503} C_VEL
LIN {X 0,Y 458.356,Z 374.18,A -85,B 0,C 180,E1 22380.114,E2 22380.114} C_VEL
LIN {X 0,Y 457.782,Z 383.751,A -85,B 0,C 180,E1 22378.41,E2 22378.41} C_VEL
LIN {X 0,Y 457.353,Z 391.275,A -85,B 0,C 180,E1 22376.629,E2 22376.629} C_VEL
LIN {X 0,Y 457.077,Z 396.706,A -85,B 0,C 180,E1 22374.878,E2 22374.878} C_VEL
LIN {X 0,Y 456.907,Z 400.627,A -85,B 0,C 180,E1 22373.001,E2 22373.001} C_VEL
LIN {X 0,Y 456.826,Z 402.733,A -85,B 0,C 180,E1 22371.085,E2 22371.085} C_VEL
LIN {X 0,Y 456.845,Z 403.108,A -85,B 0,C 180,E1 22369.224,E2 22369.224} C_VEL
LIN {X 0,Y 456.946,Z 401.649,A -85,B 0,C 180,E1 22367.287,E2 22367.287} C_VEL
LIN {X 0,Y 457.157,Z 398.454,A -85,B 0,C 180,E1 22365.407,E2 22365.407} C_VEL
LIN {X 0,Y 457.497,Z 393.198,A -85,B 0,C 180,E1 22363.482,E2 22363.482} C_VEL
LIN {X 0,Y 457.965,Z 386.231,A -85,B 0,C 180,E1 22361.696,E2 22361.696} C_VEL
LIN {X 0,Y 458.557,Z 377.821,A -85,B 0,C 180,E1 22360.063,E2 22360.063} C_VEL
LIN {X 0,Y 459.287,Z 367.511,A -85,B 0,C 180,E1 22358.508,E2 22358.508} C_VEL
LIN {X 0,Y 460.021,Z 356.188,A -85,B 0,C 180,E1 22357.174,E2 22357.174} C_VEL
LIN {X 0,Y 460.78,Z 343.789,A -85,B 0,C 180,E1 22356.019,E2 22356.019} C_VEL
LIN {X 0,Y 461.529,Z 329.145,A -85,B 0,C 180,E1 22354.972,E2 22354.972} C_VEL
LIN {X 0,Y 462.108,Z 314.306,A -85,B 0,C 180,E1 22354.196,E2 22354.196} C_VEL
LIN {X 0,Y 462.506,Z 299.307,A -85,B 0,C 180,E1 22353.653,E2 22353.653} C_VEL
LIN {X 0,Y 462.883,Z 277.523,A -85,B 0,C 180,E1 22353.195,E2 22353.195} C_VEL
LIN {X 0,Y 464.386,Z 192.861,A -85,B 0,C 180,E1 22351.633,E2 22351.633} C_VEL
LIN {X 0,Y 460.925,Z 173.887,A -85,B 0,C 180,E1 22351.035,E2 22351.035} C_VEL
LIN {X 0,Y 462.639,Z 144.306,A -85,B 0,C 180,E1 22347.131,E2 22347.131} C_VEL
LIN {X 0,Y 464.599,Z 116.036,A -85,B 0,C 180,E1 22343.328,E2 22343.328} C_VEL
LIN {X 0,Y 466.034,Z 95.182,A -85,B 0,C 180,E1 22340.47,E2 22340.47} C_VEL
LIN {X 0,Y 461.687,Z 79.522,A -85,B 0,C 180,E1 22337.78,E2 22337.78} C_VEL
LIN {X 0,Y 457.05,Z 65.007,A -85,B 0,C 180,E1 22335.049,E2 22335.049} C_VEL
LIN {X 0,Y 457.036,Z 64.863,A -85,B 0,C 180,E1 22331.452,E2 22331.452} C_VEL
LIN {X 0,Y 457.051,Z 64.869,A -85,B 0,C 180,E1 22327.796,E2 22327.796} C_VEL
LIN {X 0,Y 457.067,Z 64.865,A -85,B 0,C 180,E1 22324.14,E2 22324.14} C_VEL
LIN {X 0,Y 457.08,Z 64.864,A -85,B 0,C 180,E1 22320.376,E2 22320.376} C_VEL
LIN {X 0,Y 457.061,Z 64.866,A -85,B 0,C 180,E1 22316.614,E2 22316.614} C_VEL
LIN {X 0,Y 457.039,Z 64.867,A -85,B 0,C 180,E1 22312.963,E2 22312.963} C_VEL
LIN {X 0,Y 457.02,Z 64.867,A -85,B 0,C 180,E1 22309.411,E2 22309.411} C_VEL
LIN {X 0,Y 457.016,Z 64.866,A -85,B 0,C 180,E1 22305.687,E2 22305.687} C_VEL
LIN {X 0,Y 457.02,Z 64.865,A -85,B 0,C 180,E1 22302.033,E2 22302.033} C_VEL
LIN {X 0,Y 457.039,Z 64.868,A -85,B 0,C 180,E1 22298.437,E2 22298.437} C_VEL
LIN {X 0,Y 457.06,Z 64.864,A -85,B 0,C 180,E1 22294.888,E2 22294.888} C_VEL
LIN {X 0,Y 457.042,Z 64.866,A -85,B 0,C 180,E1 22291.231,E2 22291.231} C_VEL
LIN {X 0,Y 457.012,Z 64.869,A -85,B 0,C 180,E1 22287.736,E2 22287.736} C_VEL
LIN {X 0,Y 457.004,Z 64.869,A -85,B 0,C 180,E1 22284.048,E2 22284.048} C_VEL
LIN {X 0,Y 457.003,Z 64.872,A -85,B 0,C 180,E1 22280.294,E2 22280.294} C_VEL
LIN {X 0,Y 457.021,Z 64.868,A -85,B 0,C 180,E1 22276.764,E2 22276.764} C_VEL
LIN {X 0,Y 457.053,Z 64.862,A -85,B 0,C 180,E1 22273.214,E2 22273.214} C_VEL
LIN {X 0,Y 457.051,Z 64.863,A -85,B 0,C 180,E1 22269.539,E2 22269.539} C_VEL
LIN {X 0,Y 457.073,Z 65.267,A -85,B 0,C 180,E1 22268.747,E2 22268.747} C_VEL
LIN {X 0,Y 463.116,Z 81.187,A -85,B 0,C 180,E1 22266.361,E2 22266.361} C_VEL
LIN {X 0,Y 469.032,Z 98.91,A -85,B 0,C 180,E1 22264.007,E2 22264.007} C_VEL
LIN {X 0,Y 465.617,Z 140.662,A -85,B 0,C 180,E1 22260.165,E2 22260.165} C_VEL
LIN {X 0,Y 464.37,Z 160.528,A -85,B 0,C 180,E1 22258.418,E2 22258.418} C_VEL
LIN {X 0,Y 466.25,Z 178.05,A -85,B 0,C 180,E1 22258.017,E2 22258.017} C_VEL
LIN {X 0,Y 464.27,Z 359.701,A -85,B 0,C 180,E1 22255.181,E2 22255.181} C_VEL
LIN {X 0,Y 463.579,Z 378.325,A -85,B 0,C 180,E1 22254.672,E2 22254.672} C_VEL
LIN {X 0,Y 462.699,Z 395.895,A -85,B 0,C 180,E1 22253.97,E2 22253.97} C_VEL
LIN {X 0,Y 461.729,Z 412.721,A -85,B 0,C 180,E1 22253.076,E2 22253.076} C_VEL
LIN {X 0,Y 460.64,Z 429.791,A -85,B 0,C 180,E1 22251.922,E2 22251.922} C_VEL
LIN {X 0,Y 459.518,Z 446.601,A -85,B 0,C 180,E1 22250.507,E2 22250.507} C_VEL
LIN {X 0,Y 458.53,Z 461.634,A -85,B 0,C 180,E1 22248.96,E2 22248.96} C_VEL
LIN {X 0,Y 457.682,Z 475.787,A -85,B 0,C 180,E1 22247.202,E2 22247.202} C_VEL
LIN {X 0,Y 457.032,Z 488.171,A -85,B 0,C 180,E1 22245.351,E2 22245.351} C_VEL
LIN {X 0,Y 456.593,Z 499.552,A -85,B 0,C 180,E1 22243.294,E2 22243.294} C_VEL
LIN {X 0,Y 456.341,Z 509.296,A -85,B 0,C 180,E1 22241.118,E2 22241.118} C_VEL
LIN {X 0,Y 456.29,Z 517.005,A -85,B 0,C 180,E1 22238.951,E2 22238.951} C_VEL
LIN {X 0,Y 456.331,Z 522.903,A -85,B 0,C 180,E1 22236.796,E2 22236.796} C_VEL
LIN {X 0,Y 456.417,Z 527.3,A -85,B 0,C 180,E1 22234.524,E2 22234.524} C_VEL
LIN {X 0,Y 456.496,Z 529.925,A -85,B 0,C 180,E1 22232.26,E2 22232.26} C_VEL
LIN {X 0,Y 456.535,Z 530.832,A -85,B 0,C 180,E1 22230.001,E2 22230.001} C_VEL
LIN {X 0,Y 456.484,Z 530.023,A -85,B 0,C 180,E1 22227.741,E2 22227.741} C_VEL
LIN {X 0,Y 456.393,Z 527.408,A -85,B 0,C 180,E1 22225.42,E2 22225.42} C_VEL
LIN {X 0,Y 456.299,Z 522.887,A -85,B 0,C 180,E1 22223.079,E2 22223.079} C_VEL
LIN {X 0,Y 456.262,Z 516.999,A -85,B 0,C 180,E1 22220.923,E2 22220.923} C_VEL
LIN {X 0,Y 456.335,Z 509.276,A -85,B 0,C 180,E1 22218.756,E2 22218.756} C_VEL
LIN {X 0,Y 456.588,Z 500.142,A -85,B 0,C 180,E1 22216.708,E2 22216.708} C_VEL
LIN {X 0,Y 457.048,Z 488.864,A -85,B 0,C 180,E1 22214.652,E2 22214.652} C_VEL
LIN {X 0,Y 457.697,Z 476.936,A -85,B 0,C 180,E1 22212.849,E2 22212.849} C_VEL
LIN {X 0,Y 458.526,Z 463.474,A -85,B 0,C 180,E1 22211.152,E2 22211.152} C_VEL
LIN {X 0,Y 459.492,Z 448.94,A -85,B 0,C 180,E1 22209.626,E2 22209.626} C_VEL
LIN {X 0,Y 460.542,Z 433.337,A -85,B 0,C 180,E1 22208.276,E2 22208.276} C_VEL
LIN {X 0,Y 461.599,Z 416.923,A -85,B 0,C 180,E1 22207.121,E2 22207.121} C_VEL
LIN {X 0,Y 462.662,Z 399.023,A -85,B 0,C 180,E1 22206.131,E2 22206.131} C_VEL
LIN {X 0,Y 463.589,Z 380.464,A -85,B 0,C 180,E1 22205.366,E2 22205.366} C_VEL
LIN {X 0,Y 464.283,Z 361.793,A -85,B 0,C 180,E1 22204.839,E2 22204.839} C_VEL
LIN {X 0,Y 464.71,Z 327.32,A -85,B 0,C 180,E1 22204.275,E2 22204.275} C_VEL
LIN {X 0,Y 466.256,Z 166.043,A -85,B 0,C 180,E1 22201.768,E2 22201.768} C_VEL
LIN {X 0,Y 465.729,Z 155.672,A -85,B 0,C 180,E1 22201.538,E2 22201.538} C_VEL
LIN {X 0,Y 468.544,Z 94.215,A -85,B 0,C 180,E1 22198.318,E2 22198.318} C_VEL
LIN {X 0,Y 457.91,Z 67.56,A -85,B 0,C 180,E1 22196.072,E2 22196.072} C_VEL
LIN {X 0,Y 457.133,Z 65.265,A -85,B 0,C 180,E1 22195.834,E2 22195.834} C_VEL
LIN {X 0,Y 457.071,Z 64.865,A -85,B 0,C 180,E1 22195.49,E2 22195.49} C_VEL
LIN {X 0,Y 457.075,Z 64.862,A -85,B 0,C 180,E1 22191.75,E2 22191.75} C_VEL
LIN {X 0,Y 457.072,Z 64.862,A -85,B 0,C 180,E1 22187.983,E2 22187.983} C_VEL
LIN {X 0,Y 457.072,Z 64.864,A -85,B 0,C 180,E1 22184.252,E2 22184.252} C_VEL
LIN {X 0,Y 457.075,Z 64.859,A -85,B 0,C 180,E1 22180.518,E2 22180.518} C_VEL
LIN {X 0,Y 457.074,Z 64.861,A -85,B 0,C 180,E1 22176.812,E2 22176.812} C_VEL
LIN {X 0,Y 457.069,Z 64.861,A -85,B 0,C 180,E1 22173.092,E2 22173.092} C_VEL
LIN {X 0,Y 457.059,Z 64.861,A -85,B 0,C 180,E1 22169.468,E2 22169.468} C_VEL
LIN {X 0,Y 457.055,Z 64.864,A -85,B 0,C 180,E1 22165.806,E2 22165.806} C_VEL
LIN {X 0,Y 457.061,Z 64.865,A -85,B 0,C 180,E1 22162.102,E2 22162.102} C_VEL
LIN {X 0,Y 457.065,Z 64.86,A -85,B 0,C 180,E1 22158.361,E2 22158.361} C_VEL
LIN {X 0,Y 457.081,Z 64.857,A -85,B 0,C 180,E1 22154.699,E2 22154.699} C_VEL
LIN {X 0,Y 457.076,Z 64.863,A -85,B 0,C 180,E1 22150.971,E2 22150.971} C_VEL
LIN {X 0,Y 457.081,Z 64.859,A -85,B 0,C 180,E1 22147.289,E2 22147.289} C_VEL
LIN {X 0,Y 457.067,Z 64.856,A -85,B 0,C 180,E1 22143.511,E2 22143.511} C_VEL
LIN {X 0,Y 457.05,Z 64.854,A -85,B 0,C 180,E1 22139.874,E2 22139.874} C_VEL
LIN {X 0,Y 457.043,Z 64.861,A -85,B 0,C 180,E1 22136.237,E2 22136.237} C_VEL
LIN {X 0,Y 457.04,Z 64.864,A -85,B 0,C 180,E1 22132.457,E2 22132.457} C_VEL
LIN {X 0,Y 457.046,Z 64.865,A -85,B 0,C 180,E1 22128.772,E2 22128.772} C_VEL
LIN {X 0,Y 457.065,Z 64.861,A -85,B 0,C 180,E1 22125.17,E2 22125.17} C_VEL
LIN {X 0,Y 457.076,Z 64.857,A -85,B 0,C 180,E1 22121.507,E2 22121.507} C_VEL
LIN {X 0,Y 457.081,Z 64.85,A -85,B 0,C 180,E1 22117.763,E2 22117.763} C_VEL
LIN {X 0,Y 457.063,Z 64.857,A -85,B 0,C 180,E1 22114.035,E2 22114.035} C_VEL
LIN {X 0,Y 457.035,Z 64.854,A -85,B 0,C 180,E1 22110.512,E2 22110.512} C_VEL
LIN {X 0,Y 457.03,Z 64.867,A -85,B 0,C 180,E1 22106.843,E2 22106.843} C_VEL
LIN {X 0,Y 457.032,Z 64.866,A -85,B 0,C 180,E1 22103.17,E2 22103.17} C_VEL
LIN {X 0,Y 457.045,Z 64.858,A -85,B 0,C 180,E1 22099.577,E2 22099.577} C_VEL
LIN {X 0,Y 457.064,Z 64.857,A -85,B 0,C 180,E1 22095.921,E2 22095.921} C_VEL
LIN {X 0,Y 457.07,Z 64.86,A -85,B 0,C 180,E1 22092.186,E2 22092.186} C_VEL
LIN {X 0,Y 457.049,Z 64.864,A -85,B 0,C 180,E1 22088.569,E2 22088.569} C_VEL
LIN {X 0,Y 457.052,Z 65.097,A -85,B 0,C 180,E1 22087.317,E2 22087.317} C_VEL
LIN {X 0,Y 461.894,Z 82.569,A -85,B 0,C 180,E1 22085.089,E2 22085.089} C_VEL
LIN {X 0,Y 462.342,Z 86.235,A -85,B 0,C 180,E1 22084.662,E2 22084.662} C_VEL
LIN {X 0,Y 461.993,Z 118.988,A -85,B 0,C 180,E1 22081.067,E2 22081.067} C_VEL
LIN {X 0,Y 461.551,Z 152.017,A -85,B 0,C 180,E1 22077.421,E2 22077.421} C_VEL
LIN {X 0,Y 461.221,Z 184.922,A -85,B 0,C 180,E1 22073.891,E2 22073.891} C_VEL
LIN {X 0,Y 460.762,Z 188.581,A -85,B 0,C 180,E1 22073.625,E2 22073.625} C_VEL
LIN {X 0,Y 459.333,Z 193.687,A -85,B 0,C 180,E1 22073.472,E2 22073.472} C_VEL
LIN {X 0,Y 455.412,Z 206.806,A -85,B 0,C 180,E1 22073.401,E2 22073.401} C_VEL
LIN {X 0,Y 454.003,Z 217.15,A -85,B 0,C 180,E1 22073.293,E2 22073.293} C_VEL
LIN {X 0,Y 453.928,Z 219.462,A -85,B 0,C 180,E1 22073.258,E2 22073.258} C_VEL
LIN {X 0,Y 453.245,Z 302.119,A -85,B 0,C 180,E1 22071.905,E2 22071.905} C_VEL
LIN {X 0,Y 453.172,Z 316.67,A -85,B 0,C 180,E1 22071.449,E2 22071.449} C_VEL
LIN {X 0,Y 452.873,Z 331.103,A -85,B 0,C 180,E1 22070.751,E2 22070.751} C_VEL
LIN {X 0,Y 452.369,Z 344.662,A -85,B 0,C 180,E1 22069.831,E2 22069.831} C_VEL
LIN {X 0,Y 451.819,Z 356.423,A -85,B 0,C 180,E1 22068.782,E2 22068.782} C_VEL
LIN {X 0,Y 451.232,Z 367.393,A -85,B 0,C 180,E1 22067.538,E2 22067.538} C_VEL
LIN {X 0,Y 450.562,Z 378.104,A -85,B 0,C 180,E1 22065.971,E2 22065.971} C_VEL
LIN {X 0,Y 449.98,Z 386.938,A -85,B 0,C 180,E1 22064.278,E2 22064.278} C_VEL
LIN {X 0,Y 449.545,Z 393.571,A -85,B 0,C 180,E1 22062.588,E2 22062.588} C_VEL
LIN {X 0,Y 449.223,Z 398.722,A -85,B 0,C 180,E1 22060.774,E2 22060.774} C_VEL
LIN {X 0,Y 449.006,Z 402.248,A -85,B 0,C 180,E1 22058.837,E2 22058.837} C_VEL
LIN {X 0,Y 448.891,Z 403.939,A -85,B 0,C 180,E1 22056.779,E2 22056.779} C_VEL
LIN {X 0,Y 448.879,Z 403.59,A -85,B 0,C 180,E1 22054.726,E2 22054.726} C_VEL
LIN {X 0,Y 448.959,Z 401.412,A -85,B 0,C 180,E1 22052.807,E2 22052.807} C_VEL
LIN {X 0,Y 449.135,Z 397.721,A -85,B 0,C 180,E1 22051.019,E2 22051.019} C_VEL
LIN {X 0,Y 449.41,Z 392.247,A -85,B 0,C 180,E1 22049.234,E2 22049.234} C_VEL
LIN {X 0,Y 449.817,Z 384.668,A -85,B 0,C 180,E1 22047.451,E2 22047.451} C_VEL
LIN {X 0,Y 450.288,Z 376.135,A -85,B 0,C 180,E1 22045.924,E2 22045.924} C_VEL
LIN {X 0,Y 450.817,Z 366.195,A -85,B 0,C 180,E1 22044.527,E2 22044.527} C_VEL
LIN {X 0,Y 451.374,Z 354.017,A -85,B 0,C 180,E1 22043.193,E2 22043.193} C_VEL
LIN {X 0,Y 451.879,Z 341.107,A -85,B 0,C 180,E1 22042.114,E2 22042.114} C_VEL
LIN {X 0,Y 452.269,Z 327.937,A -85,B 0,C 180,E1 22041.289,E2 22041.289} C_VEL
LIN {X 0,Y 452.461,Z 313.697,A -85,B 0,C 180,E1 22040.648,E2 22040.648} C_VEL
LIN {X 0,Y 452.485,Z 298.419,A -85,B 0,C 180,E1 22040.221,E2 22040.221} C_VEL
LIN {X 0,Y 453.494,Z 186.536,A -85,B 0,C 180,E1 22038.425,E2 22038.425} C_VEL
LIN {X 0,Y 454.024,Z 145.445,A -85,B 0,C 180,E1 22035.785,E2 22035.785} C_VEL
LIN {X 0,Y 454.589,Z 113.509,A -85,B 0,C 180,E1 22033.648,E2 22033.648} C_VEL
LIN {X 0,Y 455.089,Z 112.624,A -85,B 0,C 180,E1 22033.436,E2 22033.436} C_VEL
LIN {X 0,Y 457.003,Z 113.855,A -85,B 0,C 180,E1 22033.148,E2 22033.148} C_VEL
LIN {X 0,Y 454.588,Z 165.438,A -85,B 0,C 180,E1 22029.125,E2 22029.125} C_VEL
LIN {X 0,Y 454.423,Z 171.461,A -85,B 0,C 180,E1 22028.704,E2 22028.704} C_VEL
LIN {X 0,Y 455.945,Z 188.527,A -85,B 0,C 180,E1 22028.318,E2 22028.318} C_VEL
LIN {X 0,Y 454.218,Z 295.246,A -85,B 0,C 180,E1 22026.421,E2 22026.421} C_VEL
LIN {X 0,Y 453.872,Z 310.765,A -85,B 0,C 180,E1 22025.914,E2 22025.914} C_VEL
LIN {X 0,Y 453.333,Z 325.654,A -85,B 0,C 180,E1 22025.182,E2 22025.182} C_VEL
LIN {X 0,Y 452.677,Z 339.582,A -85,B 0,C 180,E1 22024.254,E2 22024.254} C_VEL
LIN {X 0,Y 451.928,Z 353.096,A -85,B 0,C 180,E1 22023.077,E2 22023.077} C_VEL
LIN {X 0,Y 451.183,Z 365.395,A -85,B 0,C 180,E1 22021.689,E2 22021.689} C_VEL
LIN {X 0,Y 450.57,Z 374.938,A -85,B 0,C 180,E1 22020.339,E2 22020.339} C_VEL
LIN {X 0,Y 449.97,Z 384.247,A -85,B 0,C 180,E1 22018.67,E2 22018.67} C_VEL
LIN {X 0,Y 449.525,Z 391.48,A -85,B 0,C 180,E1 22016.979,E2 22016.979} C_VEL
LIN {X 0,Y 449.198,Z 397.425,A -85,B 0,C 180,E1 22015.106,E2 22015.106} C_VEL
LIN {X 0,Y 448.99,Z 401.738,A -85,B 0,C 180,E1 22013.039,E2 22013.039} C_VEL
LIN {X 0,Y 448.904,Z 403.844,A -85,B 0,C 180,E1 22011.089,E2 22011.089} C_VEL
LIN {X 0,Y 448.924,Z 404.233,A -85,B 0,C 180,E1 22009.224,E2 22009.224} C_VEL
LIN {X 0,Y 449.038,Z 402.777,A -85,B 0,C 180,E1 22007.224,E2 22007.224} C_VEL
LIN {X 0,Y 449.272,Z 399.6,A -85,B 0,C 180,E1 22005.31,E2 22005.31} C_VEL
LIN {X 0,Y 449.644,Z 394.361,A -85,B 0,C 180,E1 22003.353,E2 22003.353} C_VEL
LIN {X 0,Y 450.153,Z 387.423,A -85,B 0,C 180,E1 22001.537,E2 22001.537} C_VEL
LIN {X 0,Y 450.792,Z 379.059,A -85,B 0,C 180,E1 21999.876,E2 21999.876} C_VEL
LIN {X 0,Y 451.561,Z 368.935,A -85,B 0,C 180,E1 21998.315,E2 21998.315} C_VEL
LIN {X 0,Y 452.348,Z 357.723,A -85,B 0,C 180,E1 21996.958,E2 21996.958} C_VEL
LIN {X 0,Y 453.158,Z 345.491,A -85,B 0,C 180,E1 21995.782,E2 21995.782} C_VEL
LIN {X 0,Y 453.96,Z 330.88,A -85,B 0,C 180,E1 21994.706,E2 21994.706} C_VEL
LIN {X 0,Y 454.572,Z 316.694,A -85,B 0,C 180,E1 21993.928,E2 21993.928} C_VEL
LIN {X 0,Y 455.043,Z 301.258,A -85,B 0,C 180,E1 21993.331,E2 21993.331} C_VEL
LIN {X 0,Y 455.423,Z 280.634,A -85,B 0,C 180,E1 21992.87,E2 21992.87} C_VEL
LIN {X 0,Y 457.101,Z 194.053,A -85,B 0,C 180,E1 21991.235,E2 21991.235} C_VEL
LIN {X 0,Y 453.422,Z 173.746,A -85,B 0,C 180,E1 21990.572,E2 21990.572} C_VEL
LIN {X 0,Y 455.322,Z 143.693,A -85,B 0,C 180,E1 21986.544,E2 21986.544} C_VEL
LIN {X 0,Y 457.396,Z 115.594,A -85,B 0,C 180,E1 21982.708,E2 21982.708} C_VEL
LIN {X 0,Y 458.751,Z 98.16,A -85,B 0,C 180,E1 21980.276,E2 21980.276} C_VEL
LIN {X 0,Y 454.284,Z 81.866,A -85,B 0,C 180,E1 21977.418,E2 21977.418} C_VEL
LIN {X 0,Y 449.756,Z 68.186,A -85,B 0,C 180,E1 21974.813,E2 21974.813} C_VEL
LIN {X 0,Y 449.141,Z 65.941,A -85,B 0,C 180,E1 21974.306,E2 21974.306} C_VEL
LIN {X 0,Y 449.107,Z 65.853,A -85,B 0,C 180,E1 21970.649,E2 21970.649} C_VEL
LIN {X 0,Y 449.09,Z 65.856,A -85,B 0,C 180,E1 21967.034,E2 21967.034} C_VEL
LIN {X 0,Y 449.087,Z 65.857,A -85,B 0,C 180,E1 21963.319,E2 21963.319} C_VEL
LIN {X 0,Y 449.088,Z 65.856,A -85,B 0,C 180,E1 21959.618,E2 21959.618} C_VEL
LIN {X 0,Y 449.105,Z 65.855,A -85,B 0,C 180,E1 21956.043,E2 21956.043} C_VEL
LIN {X 0,Y 449.136,Z 65.852,A -85,B 0,C 180,E1 21952.453,E2 21952.453} C_VEL
LIN {X 0,Y 449.124,Z 65.856,A -85,B 0,C 180,E1 21948.702,E2 21948.702} C_VEL
LIN {X 0,Y 449.101,Z 65.854,A -85,B 0,C 180,E1 21945.034,E2 21945.034} C_VEL
LIN {X 0,Y 449.081,Z 65.853,A -85,B 0,C 180,E1 21941.435,E2 21941.435} C_VEL
LIN {X 0,Y 449.071,Z 65.856,A -85,B 0,C 180,E1 21937.759,E2 21937.759} C_VEL
LIN {X 0,Y 449.073,Z 65.858,A -85,B 0,C 180,E1 21933.984,E2 21933.984} C_VEL
LIN {X 0,Y 449.081,Z 65.858,A -85,B 0,C 180,E1 21930.378,E2 21930.378} C_VEL
LIN {X 0,Y 449.104,Z 65.858,A -85,B 0,C 180,E1 21926.792,E2 21926.792} C_VEL
LIN {X 0,Y 449.113,Z 65.858,A -85,B 0,C 180,E1 21923.051,E2 21923.051} C_VEL
LIN {X 0,Y 449.102,Z 65.857,A -85,B 0,C 180,E1 21919.393,E2 21919.393} C_VEL
LIN {X 0,Y 449.076,Z 65.853,A -85,B 0,C 180,E1 21915.802,E2 21915.802} C_VEL
LIN {X 0,Y 449.067,Z 65.863,A -85,B 0,C 180,E1 21912.147,E2 21912.147} C_VEL
LIN {X 0,Y 449.154,Z 66.123,A -85,B 0,C 180,E1 21909.503,E2 21909.503} C_VEL
LIN {X 0,Y 455.319,Z 82.499,A -85,B 0,C 180,E1 21906.934,E2 21906.934} C_VEL
LIN {X 0,Y 461.224,Z 99.877,A -85,B 0,C 180,E1 21904.535,E2 21904.535} C_VEL
LIN {X 0,Y 461.77,Z 102.118,A -85,B 0,C 180,E1 21904.262,E2 21904.262} C_VEL
LIN {X 0,Y 458.05,Z 144.537,A -85,B 0,C 180,E1 21900.281,E2 21900.281} C_VEL
LIN {X 0,Y 456.978,Z 160.758,A -85,B 0,C 180,E1 21898.835,E2 21898.835} C_VEL
LIN {X 0,Y 458.941,Z 178.835,A -85,B 0,C 180,E1 21898.411,E2 21898.411} C_VEL
LIN {X 0,Y 456.818,Z 359.137,A -85,B 0,C 180,E1 21895.552,E2 21895.552} C_VEL
LIN {X 0,Y 456.084,Z 377.711,A -85,B 0,C 180,E1 21895.036,E2 21895.036} C_VEL
LIN {X 0,Y 455.15,Z 395.234,A -85,B 0,C 180,E1 21894.324,E2 21894.324} C_VEL
LIN {X 0,Y 454.044,Z 413.054,A -85,B 0,C 180,E1 21893.353,E2 21893.353} C_VEL
LIN {X 0,Y 452.833,Z 430.734,A -85,B 0,C 180,E1 21892.116,E2 21892.116} C_VEL
LIN {X 0,Y 451.703,Z 446.514,A -85,B 0,C 180,E1 21890.743,E2 21890.743} C_VEL
LIN {X 0,Y 450.654,Z 461.392,A -85,B 0,C 180,E1 21889.17,E2 21889.17} C_VEL
LIN {X 0,Y 449.756,Z 475.395,A -85,B 0,C 180,E1 21887.386,E2 21887.386} C_VEL
LIN {X 0,Y 449.04,Z 488.33,A -85,B 0,C 180,E1 21885.39,E2 21885.39} C_VEL
LIN {X 0,Y 448.59,Z 499.556,A -85,B 0,C 180,E1 21883.273,E2 21883.273} C_VEL
LIN {X 0,Y 448.353,Z 508.849,A -85,B 0,C 180,E1 21881.119,E2 21881.119} C_VEL
LIN {X 0,Y 448.318,Z 516.595,A -85,B 0,C 180,E1 21878.853,E2 21878.853} C_VEL
LIN {X 0,Y 448.38,Z 522.307,A -85,B 0,C 180,E1 21876.66,E2 21876.66} C_VEL
LIN {X 0,Y 448.481,Z 526.349,A -85,B 0,C 180,E1 21874.476,E2 21874.476} C_VEL
LIN {X 0,Y 448.575,Z 528.891,A -85,B 0,C 180,E1 21872.173,E2 21872.173} C_VEL
LIN {X 0,Y 448.608,Z 529.709,A -85,B 0,C 180,E1 21869.873,E2 21869.873} C_VEL
LIN {X 0,Y 448.55,Z 528.81,A -85,B 0,C 180,E1 21867.574,E2 21867.574} C_VEL
LIN {X 0,Y 448.449,Z 526.179,A -85,B 0,C 180,E1 21865.269,E2 21865.269} C_VEL
LIN {X 0,Y 448.333,Z 521.717,A -85,B 0,C 180,E1 21862.942,E2 21862.942} C_VEL
LIN {X 0,Y 448.282,Z 515.836,A -85,B 0,C 180,E1 21860.76,E2 21860.76} C_VEL
LIN {X 0,Y 448.359,Z 508.076,A -85,B 0,C 180,E1 21858.553,E2 21858.553} C_VEL
LIN {X 0,Y 448.633,Z 498.895,A -85,B 0,C 180,E1 21856.468,E2 21856.468} C_VEL
LIN {X 0,Y 449.087,Z 488.364,A -85,B 0,C 180,E1 21854.505,E2 21854.505} C_VEL
LIN {X 0,Y 449.823,Z 475.567,A -85,B 0,C 180,E1 21852.539,E2 21852.539} C_VEL
LIN {X 0,Y 450.741,Z 461.624,A -85,B 0,C 180,E1 21850.768,E2 21850.768} C_VEL
LIN {X 0,Y 451.856,Z 445.971,A -85,B 0,C 180,E1 21849.131,E2 21849.131} C_VEL
LIN {X 0,Y 453.031,Z 429.641,A -85,B 0,C 180,E1 21847.738,E2 21847.738} C_VEL
LIN {X 0,Y 454.169,Z 412.868,A -85,B 0,C 180,E1 21846.587,E2 21846.587} C_VEL
LIN {X 0,Y 455.233,Z 395.362,A -85,B 0,C 180,E1 21845.648,E2 21845.648} C_VEL
LIN {X 0,Y 456.187,Z 376.818,A -85,B 0,C 180,E1 21844.912,E2 21844.912} C_VEL
LIN {X 0,Y 456.878,Z 357.753,A -85,B 0,C 180,E1 21844.41,E2 21844.41} C_VEL
LIN {X 0,Y 458.909,Z 167.165,A -85,B 0,C 180,E1 21841.4,E2 21841.4} C_VEL
LIN {X 0,Y 458.337,Z 155.713,A -85,B 0,C 180,E1 21841.143,E2 21841.143} C_VEL
LIN {X 0,Y 461.282,Z 96.819,A -85,B 0,C 180,E1 21838.001,E2 21838.001} C_VEL
LIN {X 0,Y 450.189,Z 68.943,A -85,B 0,C 180,E1 21835.598,E2 21835.598} C_VEL
LIN {X 0,Y 449.185,Z 66.238,A -85,B 0,C 180,E1 21835.305,E2 21835.305} C_VEL
LIN {X 0,Y 449.127,Z 65.852,A -85,B 0,C 180,E1 21834.947,E2 21834.947} C_VEL
LIN {X 0,Y 449.123,Z 65.854,A -85,B 0,C 180,E1 21831.186,E2 21831.186} C_VEL
LIN {X 0,Y 449.126,Z 65.855,A -85,B 0,C 180,E1 21827.41,E2 21827.41} C_VEL
LIN {X 0,Y 449.127,Z 65.851,A -85,B 0,C 180,E1 21823.64,E2 21823.64} C_VEL
LIN {X 0,Y 449.132,Z 65.855,A -85,B 0,C 180,E1 21819.877,E2 21819.877} C_VEL
LIN {X 0,Y 449.132,Z 65.851,A -85,B 0,C 180,E1 21816.091,E2 21816.091} C_VEL
LIN {X 0,Y 449.135,Z 65.849,A -85,B 0,C 180,E1 21812.295,E2 21812.295} C_VEL
LIN {X 0,Y 449.139,Z 65.85,A -85,B 0,C 180,E1 21808.596,E2 21808.596} C_VEL
LIN {X 0,Y 449.137,Z 65.85,A -85,B 0,C 180,E1 21804.882,E2 21804.882} C_VEL
LIN {X 0,Y 449.137,Z 65.849,A -85,B 0,C 180,E1 21801.135,E2 21801.135} C_VEL
LIN {X 0,Y 449.125,Z 65.849,A -85,B 0,C 180,E1 21797.356,E2 21797.356} C_VEL
LIN {X 0,Y 449.115,Z 65.846,A -85,B 0,C 180,E1 21793.65,E2 21793.65} C_VEL
LIN {X 0,Y 449.109,Z 65.845,A -85,B 0,C 180,E1 21790,E2 21790} C_VEL
LIN {X 0,Y 449.109,Z 65.85,A -85,B 0,C 180,E1 21786.263,E2 21786.263} C_VEL
LIN {X 0,Y 449.116,Z 65.854,A -85,B 0,C 180,E1 21782.552,E2 21782.552} C_VEL
LIN {X 0,Y 449.127,Z 65.849,A -85,B 0,C 180,E1 21778.852,E2 21778.852} C_VEL
LIN {X 0,Y 449.134,Z 65.846,A -85,B 0,C 180,E1 21775.147,E2 21775.147} C_VEL
LIN {X 0,Y 449.14,Z 65.851,A -85,B 0,C 180,E1 21771.422,E2 21771.422} C_VEL
LIN {X 0,Y 449.133,Z 65.851,A -85,B 0,C 180,E1 21767.66,E2 21767.66} C_VEL
LIN {X 0,Y 449.118,Z 65.851,A -85,B 0,C 180,E1 21763.975,E2 21763.975} C_VEL
LIN {X 0,Y 449.103,Z 65.852,A -85,B 0,C 180,E1 21760.341,E2 21760.341} C_VEL
LIN {X 0,Y 449.093,Z 65.83,A -85,B 0,C 180,E1 21756.653,E2 21756.653} C_VEL
LIN {X 0,Y 449.096,Z 65.854,A -85,B 0,C 180,E1 21752.844,E2 21752.844} C_VEL
LIN {X 0,Y 449.1,Z 65.841,A -85,B 0,C 180,E1 21749.198,E2 21749.198} C_VEL
LIN {X 0,Y 449.117,Z 65.846,A -85,B 0,C 180,E1 21745.564,E2 21745.564} C_VEL
LIN {X 0,Y 449.131,Z 65.857,A -85,B 0,C 180,E1 21741.797,E2 21741.797} C_VEL
LIN {X 0,Y 449.135,Z 65.853,A -85,B 0,C 180,E1 21738.032,E2 21738.032} C_VEL
LIN {X 0,Y 449.131,Z 65.856,A -85,B 0,C 180,E1 21734.205,E2 21734.205} C_VEL
LIN {X 0,Y 449.11,Z 65.851,A -85,B 0,C 180,E1 21730.546,E2 21730.546} C_VEL
LIN {X 0,Y 449.129,Z 66.088,A -85,B 0,C 180,E1 21727.747,E2 21727.747} C_VEL
LIN {X 0,Y 454.151,Z 83.816,A -85,B 0,C 180,E1 21725.452,E2 21725.452} C_VEL
LIN {X 0,Y 454.88,Z 88.197,A -85,B 0,C 180,E1 21724.926,E2 21724.926} C_VEL
LIN {X 0,Y 454.484,Z 121.279,A -85,B 0,C 180,E1 21721.277,E2 21721.277} C_VEL
LIN {X 0,Y 454.013,Z 154.329,A -85,B 0,C 180,E1 21717.617,E2 21717.617} C_VEL
LIN {X 0,Y 453.657,Z 188.712,A -85,B 0,C 180,E1 21713.923,E2 21713.923} C_VEL
LIN {X 0,Y 453.779,Z 191.134,A -85,B 0,C 180,E1 21713.736,E2 21713.736} C_VEL
LIN {X 0,Y 454.197,Z 196.201,A -85,B 0,C 180,E1 21713.631,E2 21713.631} C_VEL
LIN {X 0,Y 453.928,Z 219.462,A -85,B 0,C 180,E1 21713.258,E2 21713.258} C_VEL
LIN {X 0,Y 452.907,Z 227.133,A -85,B 0,C 180,E1 21713.178,E2 21713.178} C_VEL
LIN {X 0,Y 446.798,Z 247.476,A -85,B 0,C 180,E1 21713.119,E2 21713.119} C_VEL
LIN {X 0,Y 445.99,Z 254.063,A -85,B 0,C 180,E1 21713.046,E2 21713.046} C_VEL
LIN {X 0,Y 445.676,Z 303.891,A -85,B 0,C 180,E1 21712.197,E2 21712.197} C_VEL
LIN {X 0,Y 445.584,Z 318.243,A -85,B 0,C 180,E1 21711.729,E2 21711.729} C_VEL
LIN {X 0,Y 445.281,Z 331.949,A -85,B 0,C 180,E1 21711.054,E2 21711.054} C_VEL
LIN {X 0,Y 444.745,Z 345.587,A -85,B 0,C 180,E1 21710.117,E2 21710.117} C_VEL
LIN {X 0,Y 444.129,Z 357.922,A -85,B 0,C 180,E1 21708.995,E2 21708.995} C_VEL
LIN {X 0,Y 443.491,Z 368.885,A -85,B 0,C 180,E1 21707.718,E2 21707.718} C_VEL
LIN {X 0,Y 442.829,Z 378.721,A -85,B 0,C 180,E1 21706.258,E2 21706.258} C_VEL
LIN {X 0,Y 442.208,Z 387.4,A -85,B 0,C 180,E1 21704.593,E2 21704.593} C_VEL
LIN {X 0,Y 441.747,Z 393.962,A -85,B 0,C 180,E1 21702.947,E2 21702.947} C_VEL
LIN {X 0,Y 441.375,Z 399.345,A -85,B 0,C 180,E1 21701.101,E2 21701.101} C_VEL
LIN {X 0,Y 441.115,Z 403.05,A -85,B 0,C 180,E1 21699.128,E2 21699.128} C_VEL
LIN {X 0,Y 440.979,Z 404.875,A -85,B 0,C 180,E1 21697.163,E2 21697.163} C_VEL
LIN {X 0,Y 440.944,Z 404.927,A -85,B 0,C 180,E1 21695.203,E2 21695.203} C_VEL
LIN {X 0,Y 441.009,Z 403.211,A -85,B 0,C 180,E1 21693.248,E2 21693.248} C_VEL
LIN {X 0,Y 441.181,Z 399.628,A -85,B 0,C 180,E1 21691.298,E2 21691.298} C_VEL
LIN {X 0,Y 441.45,Z 394.478,A -85,B 0,C 180,E1 21689.48,E2 21689.48} C_VEL
LIN {X 0,Y 441.826,Z 387.933,A -85,B 0,C 180,E1 21687.794,E2 21687.794} C_VEL
LIN {X 0,Y 442.332,Z 379.27,A -85,B 0,C 180,E1 21686.111,E2 21686.111} C_VEL
LIN {X 0,Y 442.891,Z 369.336,A -85,B 0,C 180,E1 21684.622,E2 21684.622} C_VEL
LIN {X 0,Y 443.449,Z 358.386,A -85,B 0,C 180,E1 21683.331,E2 21683.331} C_VEL
LIN {X 0,Y 443.989,Z 345.713,A -85,B 0,C 180,E1 21682.169,E2 21682.169} C_VEL
LIN {X 0,Y 444.478,Z 331.568,A -85,B 0,C 180,E1 21681.2,E2 21681.2} C_VEL
LIN {X 0,Y 444.732,Z 316.277,A -85,B 0,C 180,E1 21680.463,E2 21680.463} C_VEL
LIN {X 0,Y 444.769,Z 300.858,A -85,B 0,C 180,E1 21680.003,E2 21680.003} C_VEL
LIN {X 0,Y 445.807,Z 187.808,A -85,B 0,C 180,E1 21678.157,E2 21678.157} C_VEL
LIN {X 0,Y 446.353,Z 149.976,A -85,B 0,C 180,E1 21675.734,E2 21675.734} C_VEL
LIN {X 0,Y 446.937,Z 119.187,A -85,B 0,C 180,E1 21673.665,E2 21673.665} C_VEL
LIN {X 0,Y 447.439,Z 118.22,A -85,B 0,C 180,E1 21673.445,E2 21673.445} C_VEL
LIN {X 0,Y 449.372,Z 119.235,A -85,B 0,C 180,E1 21673.167,E2 21673.167} C_VEL
LIN {X 0,Y 446.874,Z 170.85,A -85,B 0,C 180,E1 21669.111,E2 21669.111} C_VEL
LIN {X 0,Y 448.498,Z 189.352,A -85,B 0,C 180,E1 21668.68,E2 21668.68} C_VEL
LIN {X 0,Y 446.663,Z 295.792,A -85,B 0,C 180,E1 21666.749,E2 21666.749} C_VEL
LIN {X 0,Y 446.285,Z 311.731,A -85,B 0,C 180,E1 21666.216,E2 21666.216} C_VEL
LIN {X 0,Y 445.719,Z 326.398,A -85,B 0,C 180,E1 21665.48,E2 21665.48} C_VEL
LIN {X 0,Y 445.013,Z 340.511,A -85,B 0,C 180,E1 21664.522,E2 21664.522} C_VEL
LIN {X 0,Y 444.222,Z 354.002,A -85,B 0,C 180,E1 21663.326,E2 21663.326} C_VEL
LIN {X 0,Y 443.413,Z 366.572,A -85,B 0,C 180,E1 21661.882,E2 21661.882} C_VEL
LIN {X 0,Y 442.714,Z 376.698,A -85,B 0,C 180,E1 21660.403,E2 21660.403} C_VEL
LIN {X 0,Y 442.105,Z 385.673,A -85,B 0,C 180,E1 21658.747,E2 21658.747} C_VEL
LIN {X 0,Y 441.605,Z 393.256,A -85,B 0,C 180,E1 21656.902,E2 21656.902} C_VEL
LIN {X 0,Y 441.284,Z 398.706,A -85,B 0,C 180,E1 21655.107,E2 21655.107} C_VEL
LIN {X 0,Y 441.073,Z 402.846,A -85,B 0,C 180,E1 21653.078,E2 21653.078} C_VEL
LIN {X 0,Y 440.981,Z 404.98,A -85,B 0,C 180,E1 21651.051,E2 21651.051} C_VEL
LIN {X 0,Y 441.01,Z 405.308,A -85,B 0,C 180,E1 21649.063,E2 21649.063} C_VEL
LIN {X 0,Y 441.154,Z 403.713,A -85,B 0,C 180,E1 21646.983,E2 21646.983} C_VEL
LIN {X 0,Y 441.412,Z 400.346,A -85,B 0,C 180,E1 21645.031,E2 21645.031} C_VEL
LIN {X 0,Y 441.818,Z 395.193,A -85,B 0,C 180,E1 21643.114,E2 21643.114} C_VEL
LIN {X 0,Y 442.413,Z 387.815,A -85,B 0,C 180,E1 21641.185,E2 21641.185} C_VEL
LIN {X 0,Y 443.121,Z 379.201,A -85,B 0,C 180,E1 21639.494,E2 21639.494} C_VEL
LIN {X 0,Y 443.946,Z 369.127,A -85,B 0,C 180,E1 21637.942,E2 21637.942} C_VEL
LIN {X 0,Y 444.846,Z 357.17,A -85,B 0,C 180,E1 21636.502,E2 21636.502} C_VEL
LIN {X 0,Y 445.702,Z 344.771,A -85,B 0,C 180,E1 21635.331,E2 21635.331} C_VEL
LIN {X 0,Y 446.535,Z 330.492,A -85,B 0,C 180,E1 21634.285,E2 21634.285} C_VEL
LIN {X 0,Y 447.237,Z 314.752,A -85,B 0,C 180,E1 21633.442,E2 21633.442} C_VEL
LIN {X 0,Y 447.689,Z 299.146,A -85,B 0,C 180,E1 21632.878,E2 21632.878} C_VEL
LIN {X 0,Y 448.33,Z 268.655,A -85,B 0,C 180,E1 21632.243,E2 21632.243} C_VEL
LIN {X 0,Y 449.85,Z 195.247,A -85,B 0,C 180,E1 21630.824,E2 21630.824} C_VEL
LIN {X 0,Y 445.935,Z 173.74,A -85,B 0,C 180,E1 21630.106,E2 21630.106} C_VEL
LIN {X 0,Y 447.997,Z 143.451,A -85,B 0,C 180,E1 21625.987,E2 21625.987} C_VEL
LIN {X 0,Y 450.265,Z 115.09,A -85,B 0,C 180,E1 21622.042,E2 21622.042} C_VEL
LIN {X 0,Y 451.467,Z 101.131,A -85,B 0,C 180,E1 21620.077,E2 21620.077} C_VEL
LIN {X 0,Y 447.259,Z 85.588,A -85,B 0,C 180,E1 21617.297,E2 21617.297} C_VEL
LIN {X 0,Y 442.576,Z 71.349,A -85,B 0,C 180,E1 21614.523,E2 21614.523} C_VEL
LIN {X 0,Y 441.19,Z 66.982,A -85,B 0,C 180,E1 21613.596,E2 21613.596} C_VEL
LIN {X 0,Y 441.185,Z 66.843,A -85,B 0,C 180,E1 21609.918,E2 21609.918} C_VEL
LIN {X 0,Y 441.198,Z 66.844,A -85,B 0,C 180,E1 21606.245,E2 21606.245} C_VEL
LIN {X 0,Y 441.186,Z 66.842,A -85,B 0,C 180,E1 21602.468,E2 21602.468} C_VEL
LIN {X 0,Y 441.165,Z 66.843,A -85,B 0,C 180,E1 21598.831,E2 21598.831} C_VEL
LIN {X 0,Y 441.149,Z 66.845,A -85,B 0,C 180,E1 21595.19,E2 21595.19} C_VEL
LIN {X 0,Y 441.141,Z 66.846,A -85,B 0,C 180,E1 21591.528,E2 21591.528} C_VEL
LIN {X 0,Y 441.143,Z 66.845,A -85,B 0,C 180,E1 21587.832,E2 21587.832} C_VEL
LIN {X 0,Y 441.157,Z 66.842,A -85,B 0,C 180,E1 21584.218,E2 21584.218} C_VEL
LIN {X 0,Y 441.176,Z 66.845,A -85,B 0,C 180,E1 21580.528,E2 21580.528} C_VEL
LIN {X 0,Y 441.187,Z 66.842,A -85,B 0,C 180,E1 21576.776,E2 21576.776} C_VEL
LIN {X 0,Y 441.184,Z 66.841,A -85,B 0,C 180,E1 21572.901,E2 21572.901} C_VEL
LIN {X 0,Y 441.169,Z 66.843,A -85,B 0,C 180,E1 21569.19,E2 21569.19} C_VEL
LIN {X 0,Y 441.149,Z 66.845,A -85,B 0,C 180,E1 21565.485,E2 21565.485} C_VEL
LIN {X 0,Y 441.134,Z 66.847,A -85,B 0,C 180,E1 21561.774,E2 21561.774} C_VEL
LIN {X 0,Y 441.123,Z 66.85,A -85,B 0,C 180,E1 21558.211,E2 21558.211} C_VEL
LIN {X 0,Y 441.13,Z 66.85,A -85,B 0,C 180,E1 21554.441,E2 21554.441} C_VEL
LIN {X 0,Y 441.138,Z 66.845,A -85,B 0,C 180,E1 21550.751,E2 21550.751} C_VEL
LIN {X 0,Y 441.188,Z 67.249,A -85,B 0,C 180,E1 21550.248,E2 21550.248} C_VEL
LIN {X 0,Y 447.255,Z 82.854,A -85,B 0,C 180,E1 21547.685,E2 21547.685} C_VEL
LIN {X 0,Y 453.085,Z 99.569,A -85,B 0,C 180,E1 21545.263,E2 21545.263} C_VEL
LIN {X 0,Y 454.568,Z 104.795,A -85,B 0,C 180,E1 21544.576,E2 21544.576} C_VEL
LIN {X 0,Y 450.614,Z 146.987,A -85,B 0,C 180,E1 21540.539,E2 21540.539} C_VEL
LIN {X 0,Y 449.636,Z 160.973,A -85,B 0,C 180,E1 21539.275,E2 21539.275} C_VEL
LIN {X 0,Y 451.666,Z 179.682,A -85,B 0,C 180,E1 21538.821,E2 21538.821} C_VEL
LIN {X 0,Y 449.395,Z 358.492,A -85,B 0,C 180,E1 21535.939,E2 21535.939} C_VEL
LIN {X 0,Y 448.613,Z 377.04,A -85,B 0,C 180,E1 21535.416,E2 21535.416} C_VEL
LIN {X 0,Y 447.624,Z 394.613,A -85,B 0,C 180,E1 21534.69,E2 21534.69} C_VEL
LIN {X 0,Y 446.447,Z 412.39,A -85,B 0,C 180,E1 21533.704,E2 21533.704} C_VEL
LIN {X 0,Y 445.222,Z 429.119,A -85,B 0,C 180,E1 21532.519,E2 21532.519} C_VEL
LIN {X 0,Y 443.969,Z 445.444,A -85,B 0,C 180,E1 21531.083,E2 21531.083} C_VEL
LIN {X 0,Y 442.827,Z 460.594,A -85,B 0,C 180,E1 21529.454,E2 21529.454} C_VEL
LIN {X 0,Y 441.869,Z 474.464,A -85,B 0,C 180,E1 21527.651,E2 21527.651} C_VEL
LIN {X 0,Y 441.109,Z 487.207,A -85,B 0,C 180,E1 21525.649,E2 21525.649} C_VEL
LIN {X 0,Y 440.63,Z 498.337,A -85,B 0,C 180,E1 21523.517,E2 21523.517} C_VEL
LIN {X 0,Y 440.378,Z 507.399,A -85,B 0,C 180,E1 21521.393,E2 21521.393} C_VEL
LIN {X 0,Y 440.332,Z 515.051,A -85,B 0,C 180,E1 21519.147,E2 21519.147} C_VEL
LIN {X 0,Y 440.41,Z 520.891,A -85,B 0,C 180,E1 21516.912,E2 21516.912} C_VEL
LIN {X 0,Y 440.532,Z 525.051,A -85,B 0,C 180,E1 21514.688,E2 21514.688} C_VEL
LIN {X 0,Y 440.636,Z 527.7,A -85,B 0,C 180,E1 21512.342,E2 21512.342} C_VEL
LIN {X 0,Y 440.688,Z 528.618,A -85,B 0,C 180,E1 21510.001,E2 21510.001} C_VEL
LIN {X 0,Y 440.623,Z 527.807,A -85,B 0,C 180,E1 21507.66,E2 21507.66} C_VEL
LIN {X 0,Y 440.509,Z 525.26,A -85,B 0,C 180,E1 21505.314,E2 21505.314} C_VEL
LIN {X 0,Y 440.373,Z 520.915,A -85,B 0,C 180,E1 21502.959,E2 21502.959} C_VEL
LIN {X 0,Y 440.305,Z 514.662,A -85,B 0,C 180,E1 21500.591,E2 21500.591} C_VEL
LIN {X 0,Y 440.385,Z 506.867,A -85,B 0,C 180,E1 21498.343,E2 21498.343} C_VEL
LIN {X 0,Y 440.681,Z 497.487,A -85,B 0,C 180,E1 21496.188,E2 21496.188} C_VEL
LIN {X 0,Y 441.21,Z 486.244,A -85,B 0,C 180,E1 21494.087,E2 21494.087} C_VEL
LIN {X 0,Y 441.964,Z 474.172,A -85,B 0,C 180,E1 21492.218,E2 21492.218} C_VEL
LIN {X 0,Y 442.955,Z 460.142,A -85,B 0,C 180,E1 21490.417,E2 21490.417} C_VEL
LIN {X 0,Y 444.099,Z 445.049,A -85,B 0,C 180,E1 21488.818,E2 21488.818} C_VEL
LIN {X 0,Y 445.324,Z 428.956,A -85,B 0,C 180,E1 21487.424,E2 21487.424} C_VEL
LIN {X 0,Y 446.557,Z 411.864,A -85,B 0,C 180,E1 21486.234,E2 21486.234} C_VEL
LIN {X 0,Y 447.687,Z 394.275,A -85,B 0,C 180,E1 21485.28,E2 21485.28} C_VEL
LIN {X 0,Y 448.679,Z 375.661,A -85,B 0,C 180,E1 21484.537,E2 21484.537} C_VEL
LIN {X 0,Y 449.392,Z 356.651,A -85,B 0,C 180,E1 21484.039,E2 21484.039} C_VEL
LIN {X 0,Y 451.551,Z 167.775,A -85,B 0,C 180,E1 21481.01,E2 21481.01} C_VEL
LIN {X 0,Y 450.968,Z 155.756,A -85,B 0,C 180,E1 21480.735,E2 21480.735} C_VEL
LIN {X 0,Y 453.897,Z 99.076,A -85,B 0,C 180,E1 21477.649,E2 21477.649} C_VEL
LIN {X 0,Y 443.561,Z 73.079,A -85,B 0,C 180,E1 21475.363,E2 21475.363} C_VEL
LIN {X 0,Y 441.268,Z 67.328,A -85,B 0,C 180,E1 21474.793,E2 21474.793} C_VEL
LIN {X 0,Y 441.193,Z 66.841,A -85,B 0,C 180,E1 21474.448,E2 21474.448} C_VEL
LIN {X 0,Y 441.202,Z 66.841,A -85,B 0,C 180,E1 21470.604,E2 21470.604} C_VEL
LIN {X 0,Y 441.193,Z 66.841,A -85,B 0,C 180,E1 21466.813,E2 21466.813} C_VEL
LIN {X 0,Y 441.19,Z 66.839,A -85,B 0,C 180,E1 21463.012,E2 21463.012} C_VEL
LIN {X 0,Y 441.182,Z 66.841,A -85,B 0,C 180,E1 21459.388,E2 21459.388} C_VEL
LIN {X 0,Y 441.18,Z 66.836,A -85,B 0,C 180,E1 21455.553,E2 21455.553} C_VEL
LIN {X 0,Y 441.183,Z 66.837,A -85,B 0,C 180,E1 21451.806,E2 21451.806} C_VEL
LIN {X 0,Y 441.192,Z 66.835,A -85,B 0,C 180,E1 21448.124,E2 21448.124} C_VEL
LIN {X 0,Y 441.194,Z 66.836,A -85,B 0,C 180,E1 21444.356,E2 21444.356} C_VEL
LIN {X 0,Y 441.199,Z 66.841,A -85,B 0,C 180,E1 21440.565,E2 21440.565} C_VEL
LIN {X 0,Y 441.199,Z 66.841,A -85,B 0,C 180,E1 21436.727,E2 21436.727} C_VEL
LIN {X 0,Y 441.199,Z 66.836,A -85,B 0,C 180,E1 21432.965,E2 21432.965} C_VEL
LIN {X 0,Y 441.198,Z 66.831,A -85,B 0,C 180,E1 21429.128,E2 21429.128} C_VEL
LIN {X 0,Y 441.196,Z 66.836,A -85,B 0,C 180,E1 21425.331,E2 21425.331} C_VEL
LIN {X 0,Y 441.189,Z 66.838,A -85,B 0,C 180,E1 21421.558,E2 21421.558} C_VEL
LIN {X 0,Y 441.172,Z 66.84,A -85,B 0,C 180,E1 21417.922,E2 21417.922} C_VEL
LIN {X 0,Y 441.165,Z 66.838,A -85,B 0,C 180,E1 21414.146,E2 21414.146} C_VEL
LIN {X 0,Y 441.163,Z 66.835,A -85,B 0,C 180,E1 21410.352,E2 21410.352} C_VEL
LIN {X 0,Y 441.161,Z 66.836,A -85,B 0,C 180,E1 21406.633,E2 21406.633} C_VEL
LIN {X 0,Y 441.173,Z 66.839,A -85,B 0,C 180,E1 21403,E2 21403} C_VEL
LIN {X 0,Y 441.186,Z 66.84,A -85,B 0,C 180,E1 21399.295,E2 21399.295} C_VEL
LIN {X 0,Y 441.194,Z 66.816,A -85,B 0,C 180,E1 21395.64,E2 21395.64} C_VEL
LIN {X 0,Y 441.206,Z 66.838,A -85,B 0,C 180,E1 21391.826,E2 21391.826} C_VEL
LIN {X 0,Y 441.186,Z 66.835,A -85,B 0,C 180,E1 21388.126,E2 21388.126} C_VEL
LIN {X 0,Y 441.164,Z 66.83,A -85,B 0,C 180,E1 21384.45,E2 21384.45} C_VEL
LIN {X 0,Y 441.152,Z 66.843,A -85,B 0,C 180,E1 21380.776,E2 21380.776} C_VEL
LIN {X 0,Y 441.148,Z 66.843,A -85,B 0,C 180,E1 21377.058,E2 21377.058} C_VEL
LIN {X 0,Y 441.148,Z 66.839,A -85,B 0,C 180,E1 21373.318,E2 21373.318} C_VEL
LIN {X 0,Y 441.16,Z 66.844,A -85,B 0,C 180,E1 21369.725,E2 21369.725} C_VEL
LIN {X 0,Y 441.23,Z 67.091,A -85,B 0,C 180,E1 21368.195,E2 21368.195} C_VEL
LIN {X 0,Y 446.542,Z 85.668,A -85,B 0,C 180,E1 21365.759,E2 21365.759} C_VEL
LIN {X 0,Y 447.437,Z 90.143,A -85,B 0,C 180,E1 21365.205,E2 21365.205} C_VEL
LIN {X 0,Y 446.996,Z 123.637,A -85,B 0,C 180,E1 21361.493,E2 21361.493} C_VEL
LIN {X 0,Y 446.485,Z 157.239,A -85,B 0,C 180,E1 21357.76,E2 21357.76} C_VEL
LIN {X 0,Y 446.14,Z 191.098,A -85,B 0,C 180,E1 21354.129,E2 21354.129} C_VEL
LIN {X 0,Y 446.694,Z 196.439,A -85,B 0,C 180,E1 21353.983,E2 21353.983} C_VEL
LIN {X 0,Y 445.99,Z 254.063,A -85,B 0,C 180,E1 21353.046,E2 21353.046} C_VEL
LIN {X 0,Y 444.932,Z 261.737,A -85,B 0,C 180,E1 21352.966,E2 21352.966} C_VEL
LIN {X 0,Y 438.823,Z 282.081,A -85,B 0,C 180,E1 21352.904,E2 21352.904} C_VEL
LIN {X 0,Y 438.077,Z 288.666,A -85,B 0,C 180,E1 21352.826,E2 21352.826} C_VEL
LIN {X 0,Y 438.117,Z 308.228,A -85,B 0,C 180,E1 21352.43,E2 21352.43} C_VEL
LIN {X 0,Y 437.957,Z 323.048,A -85,B 0,C 180,E1 21351.881,E2 21351.881} C_VEL
LIN {X 0,Y 437.549,Z 337.191,A -85,B 0,C 180,E1 21351.093,E2 21351.093} C_VEL
LIN {X 0,Y 436.968,Z 349.776,A -85,B 0,C 180,E1 21350.142,E2 21350.142} C_VEL
LIN {X 0,Y 436.33,Z 361.563,A -85,B 0,C 180,E1 21348.988,E2 21348.988} C_VEL
LIN {X 0,Y 435.62,Z 372.347,A -85,B 0,C 180,E1 21347.635,E2 21347.635} C_VEL
LIN {X 0,Y 434.933,Z 381.654,A -85,B 0,C 180,E1 21346.149,E2 21346.149} C_VEL
LIN {X 0,Y 434.326,Z 389.613,A -85,B 0,C 180,E1 21344.531,E2 21344.531} C_VEL
LIN {X 0,Y 433.792,Z 396.564,A -85,B 0,C 180,E1 21342.647,E2 21342.647} C_VEL
LIN {X 0,Y 433.421,Z 401.439,A -85,B 0,C 180,E1 21340.768,E2 21340.768} C_VEL
LIN {X 0,Y 433.181,Z 404.564,A -85,B 0,C 180,E1 21338.895,E2 21338.895} C_VEL
LIN {X 0,Y 433.049,Z 406.131,A -85,B 0,C 180,E1 21336.866,E2 21336.866} C_VEL
LIN {X 0,Y 433.025,Z 405.79,A -85,B 0,C 180,E1 21334.767,E2 21334.767} C_VEL
LIN {X 0,Y 433.112,Z 403.635,A -85,B 0,C 180,E1 21332.778,E2 21332.778} C_VEL
LIN {X 0,Y 433.308,Z 399.967,A -85,B 0,C 180,E1 21330.924,E2 21330.924} C_VEL
LIN {X 0,Y 433.618,Z 394.509,A -85,B 0,C 180,E1 21329.074,E2 21329.074} C_VEL
LIN {X 0,Y 434.075,Z 386.954,A -85,B 0,C 180,E1 21327.226,E2 21327.226} C_VEL
LIN {X 0,Y 434.601,Z 378.451,A -85,B 0,C 180,E1 21325.645,E2 21325.645} C_VEL
LIN {X 0,Y 435.209,Z 368.166,A -85,B 0,C 180,E1 21324.15,E2 21324.15} C_VEL
LIN {X 0,Y 435.81,Z 356.408,A -85,B 0,C 180,E1 21322.816,E2 21322.816} C_VEL
LIN {X 0,Y 436.363,Z 343.547,A -85,B 0,C 180,E1 21321.699,E2 21321.699} C_VEL
LIN {X 0,Y 436.797,Z 330.476,A -85,B 0,C 180,E1 21320.845,E2 21320.845} C_VEL
LIN {X 0,Y 437.024,Z 316.074,A -85,B 0,C 180,E1 21320.169,E2 21320.169} C_VEL
LIN {X 0,Y 437.051,Z 300.645,A -85,B 0,C 180,E1 21319.72,E2 21319.72} C_VEL
LIN {X 0,Y 438.189,Z 188.343,A -85,B 0,C 180,E1 21317.846,E2 21317.846} C_VEL
LIN {X 0,Y 438.756,Z 150.613,A -85,B 0,C 180,E1 21315.414,E2 21315.414} C_VEL
LIN {X 0,Y 439.268,Z 124.768,A -85,B 0,C 180,E1 21313.673,E2 21313.673} C_VEL
LIN {X 0,Y 439.769,Z 123.833,A -85,B 0,C 180,E1 21313.454,E2 21313.454} C_VEL
LIN {X 0,Y 441.721,Z 124.973,A -85,B 0,C 180,E1 21313.157,E2 21313.157} C_VEL
LIN {X 0,Y 439.396,Z 170.94,A -85,B 0,C 180,E1 21309.51,E2 21309.51} C_VEL
LIN {X 0,Y 441.07,Z 190.129,A -85,B 0,C 180,E1 21309.056,E2 21309.056} C_VEL
LIN {X 0,Y 439.119,Z 296.476,A -85,B 0,C 180,E1 21307.085,E2 21307.085} C_VEL
LIN {X 0,Y 438.726,Z 312.111,A -85,B 0,C 180,E1 21306.554,E2 21306.554} C_VEL
LIN {X 0,Y 438.113,Z 327.214,A -85,B 0,C 180,E1 21305.784,E2 21305.784} C_VEL
LIN {X 0,Y 437.389,Z 340.983,A -85,B 0,C 180,E1 21304.837,E2 21304.837} C_VEL
LIN {X 0,Y 436.544,Z 354.576,A -85,B 0,C 180,E1 21303.618,E2 21303.618} C_VEL
LIN {X 0,Y 435.731,Z 366.543,A -85,B 0,C 180,E1 21302.236,E2 21302.236} C_VEL
LIN {X 0,Y 434.992,Z 376.735,A -85,B 0,C 180,E1 21300.761,E2 21300.761} C_VEL
LIN {X 0,Y 434.28,Z 386.492,A -85,B 0,C 180,E1 21298.954,E2 21298.954} C_VEL
LIN {X 0,Y 433.771,Z 393.691,A -85,B 0,C 180,E1 21297.201,E2 21297.201} C_VEL
LIN {X 0,Y 433.422,Z 399.211,A -85,B 0,C 180,E1 21295.424,E2 21295.424} C_VEL
LIN {X 0,Y 433.177,Z 403.41,A -85,B 0,C 180,E1 21293.443,E2 21293.443} C_VEL
LIN {X 0,Y 433.069,Z 405.855,A -85,B 0,C 180,E1 21291.437,E2 21291.437} C_VEL
